LIN {X -0.070,Y -172.197,Z 547.386,A 0.000,B 0.000,C 90.000,E1 249.571} C_DIS
LIN {X -0.092,Y -171.671,Z 547.382,A 0.000,B 0.000,C 90.000,E1 248.720} C_DIS
LIN {X -0.100,Y -167.896,Z 547.358,A 0.000,B 0.000,C 90.000,E1 244.409} C_DIS
LIN {X 0.066,Y -166.635,Z 547.348,A 0.000,B 0.000,C 90.000,E1 242.615} C_DIS
LIN {X -0.026,Y -162.621,Z 547.324,A 0.000,B 0.000,C 90.000,E1 238.280} C_DIS
LIN {X 0.033,Y -161.308,Z 547.314,A 0.000,B 0.000,C 90.000,E1 236.501} C_DIS
LIN {X -0.057,Y -157.304,Z 547.289,A 0.000,B 0.000,C 90.000,E1 232.110} C_DIS
LIN {X 0.095,Y -155.281,Z 547.275,A 0.000,B 0.000,C 90.000,E1 229.380} C_DIS
LIN {X 0.023,Y -151.646,Z 547.250,A 0.000,B 0.000,C 90.000,E1 224.919} C_DIS
LIN {X -0.040,Y -150.514,Z 547.240,A 0.000,B 0.000,C 90.000,E1 223.137} C_DIS
LIN {X -0.016,Y -147.239,Z 547.214,A 0.000,B 0.000,C 90.000,E1 218.588} C_DIS
LIN {X -0.050,Y -145.263,Z 547.194,A 0.000,B 0.000,C 90.000,E1 214.945} C_DIS
LIN {X -0.016,Y -142.373,Z 547.163,A 0.000,B 0.000,C 90.000,E1 209.411} C_DIS
LIN {X -0.021,Y -141.757,Z 547.153,A 0.000,B 0.000,C 90.000,E1 207.564} C_DIS
LIN {X 0.030,Y -139.498,Z 547.117,A 0.000,B 0.000,C 90.000,E1 201.046} C_DIS
LIN {X 0.066,Y -139.004,Z 547.101,A 0.000,B 0.000,C 90.000,E1 198.236} C_DIS
LIN {X 0.023,Y -138.339,Z 547.055,A 0.000,B 0.000,C 90.000,E1 189.849} C_DIS
LIN {X 0.045,Y -139.406,Z 547.008,A 0.000,B 0.000,C 90.000,E1 181.432} C_DIS
LIN {X -0.041,Y -141.314,Z 546.972,A 0.000,B 0.000,C 90.000,E1 174.951} C_DIS
LIN {X 0.057,Y -142.673,Z 546.956,A 0.000,B 0.000,C 90.000,E1 172.129} C_DIS
LIN {X 0.038,Y -145.026,Z 546.931,A 0.000,B 0.000,C 90.000,E1 167.521} C_DIS
LIN {X -0.005,Y -147.652,Z 546.910,A 0.000,B 0.000,C 90.000,E1 163.866} C_DIS
LIN {X -0.071,Y -150.288,Z 546.890,A 0.000,B 0.000,C 90.000,E1 160.242} C_DIS
LIN {X -0.058,Y -153.695,Z 546.870,A 0.000,B 0.000,C 90.000,E1 156.613} C_DIS
LIN {X -0.003,Y -157.109,Z 546.850,A 0.000,B 0.000,C 90.000,E1 152.999} C_DIS
LIN {X 0.074,Y -161.250,Z 546.830,A 0.000,B 0.000,C 90.000,E1 149.410} C_DIS
LIN {X 0.020,Y -163.336,Z 546.820,A 0.000,B 0.000,C 90.000,E1 147.661} C_DIS
LIN {X 0.026,Y -167.791,Z 546.801,A 0.000,B 0.000,C 90.000,E1 144.149} C_DIS
LIN {X 0.041,Y -171.605,Z 546.786,A 0.000,B 0.000,C 90.000,E1 141.537} C_DIS
LIN {X 0.090,Y -176.559,Z 546.767,A 0.000,B 0.000,C 90.000,E1 138.081} C_DIS
LIN {X -0.036,Y -180.857,Z 546.753,A 0.000,B 0.000,C 90.000,E1 135.567} C_DIS
LIN {X -0.052,Y -186.270,Z 546.734,A 0.000,B 0.000,C 90.000,E1 132.204} C_DIS
LIN {X 0.015,Y -191.369,Z 546.719,A 0.000,B 0.000,C 90.000,E1 129.402} C_DIS
LIN {X -0.035,Y -191.935,Z 546.717,A 0.000,B 0.000,C 90.000,E1 129.072} C_DIS
LIN {X 0.095,Y -289.045,Z 546.717,A 0.000,B 0.000,C 90.000,E1 129.036} C_DIS
LIN {X -0.010,Y -290.435,Z 546.717,A 0.000,B 0.000,C 90.000,E1 129.036} C_DIS
LIN {X 0.173,Y -294.486,Z 546.716,A 0.000,B 0.000,C 90.000,E1 128.830} C_DIS
LIN {X 0.062,Y -297.700,Z 546.714,A 0.000,B 0.000,C 90.000,E1 128.588} C_DIS
LIN {X 0.115,Y -301.387,Z 546.712,A 0.000,B 0.000,C 90.000,E1 128.096} C_DIS
LIN {X -0.126,Y -303.164,Z 546.710,A 0.000,B 0.000,C 90.000,E1 127.810} C_DIS
LIN {X 0.057,Y -304.555,Z 546.708,A 0.000,B 0.000,C 90.000,E1 127.443} C_DIS
LIN {X 0.012,Y -308.418,Z 546.701,A 0.000,B 0.000,C 90.000,E1 126.137} C_DIS
LIN {X 0.078,Y -318.623,Z 546.683,A 0.000,B 0.000,C 90.000,E1 122.880} C_DIS
LIN {X 0.153,Y -329.135,Z 546.667,A 0.000,B 0.000,C 90.000,E1 120.001} C_DIS
LIN {X 0.045,Y -341.016,Z 546.651,A 0.000,B 0.000,C 90.000,E1 117.206} C_DIS
LIN {X -0.031,Y -354.367,Z 546.636,A 0.000,B 0.000,C 90.000,E1 114.463} C_DIS
LIN {X -0.113,Y -367.569,Z 546.623,A 0.000,B 0.000,C 90.000,E1 112.078} C_DIS
LIN {X 0.070,Y -382.126,Z 546.609,A 0.000,B 0.000,C 90.000,E1 109.704} C_DIS
LIN {X 0.149,Y -398.143,Z 546.597,A 0.000,B 0.000,C 90.000,E1 107.402} C_DIS
LIN {X -0.002,Y -415.738,Z 546.584,A 0.000,B 0.000,C 90.000,E1 105.190} C_DIS
LIN {X 0.088,Y -435.005,Z 546.572,A 0.000,B 0.000,C 90.000,E1 103.008} C_DIS
LIN {X -0.087,Y -455.210,Z 546.561,A 0.000,B 0.000,C 90.000,E1 101.007} C_DIS
LIN {X -0.092,Y -475.919,Z 546.551,A 0.000,B 0.000,C 90.000,E1 99.151} C_DIS
LIN {X 0.019,Y -477.987,Z 546.550,A 0.000,B 0.000,C 90.000,E1 98.916} C_DIS
LIN {X -0.115,Y -479.747,Z 546.548,A 0.000,B 0.000,C 90.000,E1 98.681} C_DIS
LIN {X 0.155,Y -481.069,Z 546.547,A 0.000,B 0.000,C 90.000,E1 98.398} C_DIS
LIN {X -0.161,Y -482.719,Z 546.544,A 0.000,B 0.000,C 90.000,E1 97.936} C_DIS
LIN {X 0.071,Y -483.299,Z 546.541,A 0.000,B 0.000,C 90.000,E1 97.409} C_DIS
LIN {X 0.248,Y -482.905,Z 546.538,A 0.000,B 0.000,C 90.000,E1 96.891} C_DIS
LIN {X -0.050,Y -481.476,Z 546.536,A 0.000,B 0.000,C 90.000,E1 96.429} C_DIS
LIN {X -0.225,Y -480.299,Z 546.534,A 0.000,B 0.000,C 90.000,E1 96.201} C_DIS
LIN {X 0.127,Y -478.728,Z 546.533,A 0.000,B 0.000,C 90.000,E1 95.910} C_DIS
LIN {X -0.090,Y -461.364,Z 546.520,A 0.000,B 0.000,C 90.000,E1 93.669} C_DIS
LIN {X -0.033,Y -450.979,Z 546.512,A 0.000,B 0.000,C 90.000,E1 92.121} C_DIS
LIN {X -0.051,Y -437.218,Z 546.499,A 0.000,B 0.000,C 90.000,E1 89.771} C_DIS
LIN {X -0.127,Y -429.303,Z 546.491,A 0.000,B 0.000,C 90.000,E1 88.453} C_DIS
LIN {X 0.048,Y -416.530,Z 546.479,A 0.000,B 0.000,C 90.000,E1 86.274} C_DIS
LIN {X -0.049,Y -403.962,Z 546.467,A 0.000,B 0.000,C 90.000,E1 84.090} C_DIS
LIN {X 0.042,Y -391.625,Z 546.455,A 0.000,B 0.000,C 90.000,E1 81.837} C_DIS
LIN {X -0.102,Y -382.389,Z 546.445,A 0.000,B 0.000,C 90.000,E1 80.151} C_DIS
LIN {X -0.027,Y -371.645,Z 546.434,A 0.000,B 0.000,C 90.000,E1 78.117} C_DIS
LIN {X -0.023,Y -358.447,Z 546.419,A 0.000,B 0.000,C 90.000,E1 75.463} C_DIS
LIN {X -0.192,Y -348.165,Z 546.406,A 0.000,B 0.000,C 90.000,E1 73.087} C_DIS
LIN {X 0.034,Y -340.049,Z 546.394,A 0.000,B 0.000,C 90.000,E1 70.913} C_DIS
LIN {X 0.097,Y -327.539,Z 546.373,A 0.000,B 0.000,C 90.000,E1 67.177} C_DIS
LIN {X 0.041,Y -317.890,Z 546.356,A 0.000,B 0.000,C 90.000,E1 64.024} C_DIS
LIN {X 0.004,Y -310.442,Z 546.341,A 0.000,B 0.000,C 90.000,E1 61.463} C_DIS
LIN {X -0.043,Y -302.984,Z 546.327,A 0.000,B 0.000,C 90.000,E1 58.869} C_DIS
LIN {X 0.061,Y -294.026,Z 546.309,A 0.000,B 0.000,C 90.000,E1 55.548} C_DIS
LIN {X -0.050,Y -287.193,Z 546.294,A 0.000,B 0.000,C 90.000,E1 52.889} C_DIS
LIN {X -0.004,Y -282.059,Z 546.282,A 0.000,B 0.000,C 90.000,E1 50.848} C_DIS
LIN {X 0.118,Y -276.452,Z 546.271,A 0.000,B 0.000,C 90.000,E1 48.771} C_DIS
LIN {X 0.117,Y -272.330,Z 546.263,A 0.000,B 0.000,C 90.000,E1 47.391} C_DIS
LIN {X 0.127,Y -266.837,Z 546.254,A 0.000,B 0.000,C 90.000,E1 45.648} C_DIS
LIN {X 0.083,Y -259.769,Z 546.242,A 0.000,B 0.000,C 90.000,E1 43.542} C_DIS
LIN {X 0.002,Y -248.281,Z 546.222,A 0.000,B 0.000,C 90.000,E1 39.967} C_DIS
LIN {X 0.028,Y -238.665,Z 546.204,A 0.000,B 0.000,C 90.000,E1 36.664} C_DIS
LIN {X -0.074,Y -230.808,Z 546.187,A 0.000,B 0.000,C 90.000,E1 33.706} C_DIS
LIN {X -0.045,Y -223.755,Z 546.170,A 0.000,B 0.000,C 90.000,E1 30.669} C_DIS
LIN {X -0.028,Y -217.536,Z 546.153,A 0.000,B 0.000,C 90.000,E1 27.590} C_DIS
LIN {X 0.020,Y -212.107,Z 546.136,A 0.000,B 0.000,C 90.000,E1 24.463} C_DIS
LIN {X -0.036,Y -206.520,Z 546.114,A 0.000,B 0.000,C 90.000,E1 20.536} C_DIS
LIN {X -0.048,Y -202.027,Z 546.092,A 0.000,B 0.000,C 90.000,E1 16.551} C_DIS
LIN {X -0.081,Y -198.706,Z 546.070,A 0.000,B 0.000,C 90.000,E1 12.535} C_DIS
LIN {X -0.008,Y -195.844,Z 546.038,A 0.000,B 0.000,C 90.000,E1 6.834} C_DIS
LIN {X -0.024,Y -195.870,Z 545.979,A 0.000,B 0.000,C 90.000,E1 356.274} C_DIS
LIN {X 0.050,Y -198.724,Z 545.948,A 0.000,B 0.000,C 90.000,E1 350.557} C_DIS
LIN {X 0.079,Y -202.621,Z 545.921,A 0.000,B 0.000,C 90.000,E1 345.700} C_DIS
LIN {X 0.017,Y -206.754,Z 545.898,A 0.000,B 0.000,C 90.000,E1 341.710} C_DIS
LIN {X 0.012,Y -211.728,Z 545.876,A 0.000,B 0.000,C 90.000,E1 337.741} C_DIS
LIN {X -0.006,Y -217.254,Z 545.855,A 0.000,B 0.000,C 90.000,E1 333.819} C_DIS
LIN {X 0.067,Y -223.354,Z 545.833,A 0.000,B 0.000,C 90.000,E1 329.921} C_DIS
LIN {X 0.085,Y -230.113,Z 545.812,A 0.000,B 0.000,C 90.000,E1 326.087} C_DIS
LIN {X -0.001,Y -235.917,Z 545.795,A 0.000,B 0.000,C 90.000,E1 323.084} C_DIS
LIN {X -0.111,Y -243.607,Z 545.774,A 0.000,B 0.000,C 90.000,E1 319.380} C_DIS
LIN {X 0.151,Y -252.265,Z 545.754,A 0.000,B 0.000,C 90.000,E1 315.648} C_DIS
LIN {X -0.011,Y -262.199,Z 545.734,A 0.000,B 0.000,C 90.000,E1 312.081} C_DIS
LIN {X 0.031,Y -273.518,Z 545.714,A 0.000,B 0.000,C 90.000,E1 308.543} C_DIS
LIN {X -0.026,Y -286.116,Z 545.695,A 0.000,B 0.000,C 90.000,E1 305.105} C_DIS
LIN {X 0.059,Y -300.199,Z 545.676,A 0.000,B 0.000,C 90.000,E1 301.720} C_DIS
LIN {X 0.124,Y -312.274,Z 545.662,A 0.000,B 0.000,C 90.000,E1 299.077} C_DIS
LIN {X -0.142,Y -326.845,Z 545.646,A 0.000,B 0.000,C 90.000,E1 296.232} C_DIS
LIN {X -0.113,Y -339.476,Z 545.633,A 0.000,B 0.000,C 90.000,E1 294.027} C_DIS
LIN {X 0.048,Y -351.407,Z 545.623,A 0.000,B 0.000,C 90.000,E1 292.153} C_DIS
LIN {X -0.019,Y -368.800,Z 545.610,A 0.000,B 0.000,C 90.000,E1 289.758} C_DIS
LIN {X 0.098,Y -385.146,Z 545.598,A 0.000,B 0.000,C 90.000,E1 287.692} C_DIS
LIN {X -0.046,Y -402.080,Z 545.587,A 0.000,B 0.000,C 90.000,E1 285.717} C_DIS
LIN {X -0.142,Y -416.797,Z 545.578,A 0.000,B 0.000,C 90.000,E1 284.064} C_DIS
LIN {X -0.154,Y -428.707,Z 545.570,A 0.000,B 0.000,C 90.000,E1 282.703} C_DIS
LIN {X 0.133,Y -437.908,Z 545.565,A 0.000,B 0.000,C 90.000,E1 281.591} C_DIS
LIN {X -0.204,Y -444.480,Z 545.560,A 0.000,B 0.000,C 90.000,E1 280.838} C_DIS
LIN {X -0.161,Y -452.677,Z 545.554,A 0.000,B 0.000,C 90.000,E1 279.782} C_DIS
LIN {X -0.175,Y -460.261,Z 545.548,A 0.000,B 0.000,C 90.000,E1 278.746} C_DIS
LIN {X 0.149,Y -465.527,Z 545.544,A 0.000,B 0.000,C 90.000,E1 277.936} C_DIS
LIN {X 0.053,Y -470.288,Z 545.540,A 0.000,B 0.000,C 90.000,E1 277.182} C_DIS
LIN {X -0.001,Y -474.504,Z 545.536,A 0.000,B 0.000,C 90.000,E1 276.429} C_DIS
LIN {X -0.077,Y -478.274,Z 545.531,A 0.000,B 0.000,C 90.000,E1 275.682} C_DIS
LIN {X 0.068,Y -480.405,Z 545.529,A 0.000,B 0.000,C 90.000,E1 275.163} C_DIS
LIN {X 0.225,Y -482.231,Z 545.526,A 0.000,B 0.000,C 90.000,E1 274.645} C_DIS
LIN {X -0.129,Y -483.769,Z 545.523,A 0.000,B 0.000,C 90.000,E1 274.188} C_DIS
LIN {X 0.044,Y -485.000,Z 545.520,A 0.000,B 0.000,C 90.000,E1 273.669} C_DIS
LIN {X 0.196,Y -485.831,Z 545.518,A 0.000,B 0.000,C 90.000,E1 273.154} C_DIS
LIN {X -0.104,Y -486.404,Z 545.515,A 0.000,B 0.000,C 90.000,E1 272.694} C_DIS
LIN {X 0.064,Y -486.626,Z 545.512,A 0.000,B 0.000,C 90.000,E1 272.178} C_DIS
LIN {X -0.234,Y -486.498,Z 545.509,A 0.000,B 0.000,C 90.000,E1 271.718} C_DIS
LIN {X -0.061,Y -485.933,Z 545.507,A 0.000,B 0.000,C 90.000,E1 271.203} C_DIS
LIN {X 0.112,Y -484.982,Z 545.504,A 0.000,B 0.000,C 90.000,E1 270.688} C_DIS
LIN {X -0.202,Y -483.464,Z 545.501,A 0.000,B 0.000,C 90.000,E1 270.229} C_DIS
LIN {X -0.036,Y -481.307,Z 545.498,A 0.000,B 0.000,C 90.000,E1 269.714} C_DIS
LIN {X 0.119,Y -478.472,Z 545.496,A 0.000,B 0.000,C 90.000,E1 269.198} C_DIS
LIN {X -0.053,Y -476.758,Z 545.494,A 0.000,B 0.000,C 90.000,E1 268.969} C_DIS
LIN {X -0.224,Y -474.771,Z 545.493,A 0.000,B 0.000,C 90.000,E1 268.740} C_DIS
LIN {X -0.110,Y -470.060,Z 545.490,A 0.000,B 0.000,C 90.000,E1 268.224} C_DIS
LIN {X 0.194,Y -467.224,Z 545.489,A 0.000,B 0.000,C 90.000,E1 267.936} C_DIS
LIN {X 0.015,Y -464.003,Z 545.487,A 0.000,B 0.000,C 90.000,E1 267.707} C_DIS
LIN {X 0.162,Y -460.906,Z 545.486,A 0.000,B 0.000,C 90.000,E1 267.478} C_DIS
LIN {X -0.161,Y -454.171,Z 545.484,A 0.000,B 0.000,C 90.000,E1 267.135} C_DIS
LIN {X 0.082,Y -447.074,Z 545.482,A 0.000,B 0.000,C 90.000,E1 266.788} C_DIS
LIN {X -0.182,Y -439.758,Z 545.481,A 0.000,B 0.000,C 90.000,E1 266.560} C_DIS
LIN {X -0.050,Y -431.608,Z 545.480,A 0.000,B 0.000,C 90.000,E1 266.331} C_DIS
LIN {X 0.058,Y -423.111,Z 545.479,A 0.000,B 0.000,C 90.000,E1 266.159} C_DIS
LIN {X 0.085,Y -412.497,Z 545.478,A 0.000,B 0.000,C 90.000,E1 266.045} C_DIS
LIN {X -0.072,Y -404.407,Z 545.478,A 0.000,B 0.000,C 90.000,E1 266.045} C_DIS
LIN {X -0.066,Y -180.921,Z 545.478,A 0.000,B 0.000,C 90.000,E1 266.045} C_DIS
LIN {X -0.026,Y -180.862,Z 545.472,A 0.000,B 0.000,C 90.000,E1 265.008} C_DIS
LIN {X 0.054,Y -178.917,Z 545.443,A 0.000,B 0.000,C 90.000,E1 259.746} C_DIS
LIN {X -0.037,Y -175.963,Z 545.415,A 0.000,B 0.000,C 90.000,E1 254.685} C_DIS
LIN {X 0.079,Y -175.438,Z 545.410,A 0.000,B 0.000,C 90.000,E1 253.795} C_DIS
LIN {X -0.080,Y -172.196,Z 545.386,A 0.000,B 0.000,C 90.000,E1 249.571} C_DIS
LIN {X -0.101,Y -171.669,Z 545.382,A 0.000,B 0.000,C 90.000,E1 248.720} C_DIS
LIN {X 0.042,Y -167.894,Z 545.358,A 0.000,B 0.000,C 90.000,E1 244.357} C_DIS
LIN {X 0.057,Y -166.632,Z 545.348,A 0.000,B 0.000,C 90.000,E1 242.615} C_DIS
LIN {X -0.035,Y -162.618,Z 545.324,A 0.000,B 0.000,C 90.000,E1 238.280} C_DIS
LIN {X 0.023,Y -161.304,Z 545.314,A 0.000,B 0.000,C 90.000,E1 236.501} C_DIS
LIN {X -0.067,Y -157.302,Z 545.289,A 0.000,B 0.000,C 90.000,E1 232.110} C_DIS
LIN {X 0.086,Y -155.278,Z 545.275,A 0.000,B 0.000,C 90.000,E1 229.380} C_DIS
LIN {X 0.014,Y -151.643,Z 545.250,A 0.000,B 0.000,C 90.000,E1 224.919} C_DIS
LIN {X -0.049,Y -150.512,Z 545.240,A 0.000,B 0.000,C 90.000,E1 223.137} C_DIS
LIN {X -0.025,Y -147.237,Z 545.214,A 0.000,B 0.000,C 90.000,E1 218.588} C_DIS
LIN {X 0.060,Y -145.260,Z 545.194,A 0.000,B 0.000,C 90.000,E1 214.898} C_DIS
LIN {X -0.025,Y -142.371,Z 545.163,A 0.000,B 0.000,C 90.000,E1 209.411} C_DIS
LIN {X -0.030,Y -141.756,Z 545.153,A 0.000,B 0.000,C 90.000,E1 207.564} C_DIS
LIN {X 0.021,Y -139.497,Z 545.117,A 0.000,B 0.000,C 90.000,E1 201.046} C_DIS
LIN {X 0.058,Y -139.003,Z 545.101,A 0.000,B 0.000,C 90.000,E1 198.236} C_DIS
LIN {X 0.014,Y -138.339,Z 545.055,A 0.000,B 0.000,C 90.000,E1 189.849} C_DIS
LIN {X 0.036,Y -139.406,Z 545.008,A 0.000,B 0.000,C 90.000,E1 181.432} C_DIS
LIN {X -0.050,Y -141.316,Z 544.972,A 0.000,B 0.000,C 90.000,E1 174.951} C_DIS
LIN {X 0.049,Y -142.675,Z 544.956,A 0.000,B 0.000,C 90.000,E1 172.129} C_DIS
LIN {X 0.029,Y -145.028,Z 544.931,A 0.000,B 0.000,C 90.000,E1 167.521} C_DIS
LIN {X -0.014,Y -147.655,Z 544.910,A 0.000,B 0.000,C 90.000,E1 163.866} C_DIS
LIN {X 0.062,Y -150.292,Z 544.890,A 0.000,B 0.000,C 90.000,E1 160.188} C_DIS
LIN {X -0.067,Y -153.699,Z 544.870,A 0.000,B 0.000,C 90.000,E1 156.613} C_DIS
LIN {X -0.012,Y -157.113,Z 544.850,A 0.000,B 0.000,C 90.000,E1 152.999} C_DIS
LIN {X 0.064,Y -161.255,Z 544.830,A 0.000,B 0.000,C 90.000,E1 149.410} C_DIS
LIN {X -0.008,Y -164.373,Z 544.815,A 0.000,B 0.000,C 90.000,E1 146.786} C_DIS
LIN {X -0.021,Y -169.047,Z 544.796,A 0.000,B 0.000,C 90.000,E1 143.290} C_DIS
LIN {X 0.032,Y -171.609,Z 544.786,A 0.000,B 0.000,C 90.000,E1 141.537} C_DIS
LIN {X 0.080,Y -176.565,Z 544.767,A 0.000,B 0.000,C 90.000,E1 138.081} C_DIS
LIN {X -0.046,Y -180.863,Z 544.753,A 0.000,B 0.000,C 90.000,E1 135.567} C_DIS
LIN {X -0.063,Y -186.276,Z 544.734,A 0.000,B 0.000,C 90.000,E1 132.204} C_DIS
LIN {X 0.003,Y -191.374,Z 544.719,A 0.000,B 0.000,C 90.000,E1 129.402} C_DIS
LIN {X 0.026,Y -191.964,Z 544.717,A 0.000,B 0.000,C 90.000,E1 129.036} C_DIS
LIN {X 0.006,Y -288.546,Z 544.717,A 0.000,B 0.000,C 90.000,E1 129.036} C_DIS
LIN {X -0.029,Y -289.471,Z 544.717,A 0.000,B 0.000,C 90.000,E1 129.036} C_DIS
LIN {X 0.156,Y -294.233,Z 544.716,A 0.000,B 0.000,C 90.000,E1 128.830} C_DIS
LIN {X 0.062,Y -297.157,Z 544.715,A 0.000,B 0.000,C 90.000,E1 128.624} C_DIS
LIN {X 0.018,Y -300.901,Z 544.712,A 0.000,B 0.000,C 90.000,E1 128.177} C_DIS
LIN {X -0.020,Y -302.779,Z 544.710,A 0.000,B 0.000,C 90.000,E1 127.855} C_DIS
LIN {X -0.005,Y -304.248,Z 544.708,A 0.000,B 0.000,C 90.000,E1 127.523} C_DIS
LIN {X -0.032,Y -306.343,Z 544.705,A 0.000,B 0.000,C 90.000,E1 126.870} C_DIS
LIN {X 0.149,Y -316.216,Z 544.687,A 0.000,B 0.000,C 90.000,E1 123.579} C_DIS
LIN {X 0.050,Y -326.408,Z 544.671,A 0.000,B 0.000,C 90.000,E1 120.718} C_DIS
LIN {X 0.013,Y -337.944,Z 544.655,A 0.000,B 0.000,C 90.000,E1 117.897} C_DIS
LIN {X -0.160,Y -350.921,Z 544.640,A 0.000,B 0.000,C 90.000,E1 115.155} C_DIS
LIN {X 0.006,Y -363.767,Z 544.626,A 0.000,B 0.000,C 90.000,E1 112.717} C_DIS
LIN {X 0.016,Y -377.939,Z 544.613,A 0.000,B 0.000,C 90.000,E1 110.355} C_DIS
LIN {X -0.026,Y -393.541,Z 544.600,A 0.000,B 0.000,C 90.000,E1 108.055} C_DIS
LIN {X 0.091,Y -410.687,Z 544.588,A 0.000,B 0.000,C 90.000,E1 105.788} C_DIS
LIN {X 0.135,Y -429.504,Z 544.576,A 0.000,B 0.000,C 90.000,E1 103.592} C_DIS
LIN {X 0.020,Y -449.542,Z 544.564,A 0.000,B 0.000,C 90.000,E1 101.535} C_DIS
LIN {X 0.197,Y -470.144,Z 544.554,A 0.000,B 0.000,C 90.000,E1 99.613} C_DIS
LIN {X -0.175,Y -475.373,Z 544.551,A 0.000,B 0.000,C 90.000,E1 99.208} C_DIS
LIN {X -0.069,Y -477.617,Z 544.550,A 0.000,B 0.000,C 90.000,E1 98.973} C_DIS
LIN {X -0.223,Y -479.463,Z 544.548,A 0.000,B 0.000,C 90.000,E1 98.746} C_DIS
LIN {X 0.172,Y -480.860,Z 544.547,A 0.000,B 0.000,C 90.000,E1 98.454} C_DIS
LIN {X -0.147,Y -482.685,Z 544.544,A 0.000,B 0.000,C 90.000,E1 97.992} C_DIS
LIN {X 0.022,Y -483.410,Z 544.542,A 0.000,B 0.000,C 90.000,E1 97.473} C_DIS
LIN {X 0.261,Y -483.156,Z 544.539,A 0.000,B 0.000,C 90.000,E1 96.947} C_DIS
LIN {X -0.038,Y -481.887,Z 544.536,A 0.000,B 0.000,C 90.000,E1 96.486} C_DIS
LIN {X -0.213,Y -480.809,Z 544.535,A 0.000,B 0.000,C 90.000,E1 96.258} C_DIS
LIN {X 0.141,Y -479.362,Z 544.533,A 0.000,B 0.000,C 90.000,E1 95.967} C_DIS
LIN {X 0.053,Y -467.646,Z 544.525,A 0.000,B 0.000,C 90.000,E1 94.473} C_DIS
LIN {X 0.236,Y -456.621,Z 544.516,A 0.000,B 0.000,C 90.000,E1 92.922} C_DIS
LIN {X 0.201,Y -446.737,Z 544.508,A 0.000,B 0.000,C 90.000,E1 91.375} C_DIS
LIN {X 0.165,Y -436.140,Z 544.498,A 0.000,B 0.000,C 90.000,E1 89.542} C_DIS
LIN {X -0.204,Y -426.561,Z 544.489,A 0.000,B 0.000,C 90.000,E1 87.993} C_DIS
LIN {X -0.080,Y -413.840,Z 544.477,A 0.000,B 0.000,C 90.000,E1 85.812} C_DIS
LIN {X 0.166,Y -401.295,Z 544.464,A 0.000,B 0.000,C 90.000,E1 83.571} C_DIS
LIN {X 0.191,Y -390.524,Z 544.453,A 0.000,B 0.000,C 90.000,E1 81.602} C_DIS
LIN {X -0.010,Y -379.714,Z 544.442,A 0.000,B 0.000,C 90.000,E1 79.634} C_DIS
LIN {X 0.071,Y -368.956,Z 544.431,A 0.000,B 0.000,C 90.000,E1 77.589} C_DIS
LIN {X 0.087,Y -358.797,Z 544.420,A 0.000,B 0.000,C 90.000,E1 75.519} C_DIS
LIN {X 0.000,Y -349.685,Z 544.408,A 0.000,B 0.000,C 90.000,E1 73.433} C_DIS
LIN {X 0.160,Y -340.322,Z 544.394,A 0.000,B 0.000,C 90.000,E1 70.967} C_DIS
LIN {X -0.067,Y -327.793,Z 544.374,A 0.000,B 0.000,C 90.000,E1 67.283} C_DIS
LIN {X 0.052,Y -318.151,Z 544.356,A 0.000,B 0.000,C 90.000,E1 64.101} C_DIS
LIN {X -0.111,Y -310.668,Z 544.342,A 0.000,B 0.000,C 90.000,E1 61.563} C_DIS
LIN {X -0.032,Y -303.212,Z 544.327,A 0.000,B 0.000,C 90.000,E1 58.948} C_DIS
LIN {X -0.170,Y -294.218,Z 544.309,A 0.000,B 0.000,C 90.000,E1 55.674} C_DIS
LIN {X -0.038,Y -287.364,Z 544.294,A 0.000,B 0.000,C 90.000,E1 52.970} C_DIS
LIN {X 0.011,Y -282.228,Z 544.283,A 0.000,B 0.000,C 90.000,E1 50.928} C_DIS
LIN {X 0.134,Y -276.622,Z 544.272,A 0.000,B 0.000,C 90.000,E1 48.852} C_DIS
LIN {X 0.134,Y -272.512,Z 544.264,A 0.000,B 0.000,C 90.000,E1 47.472} C_DIS
LIN {X 0.028,Y -265.856,Z 544.252,A 0.000,B 0.000,C 90.000,E1 45.405} C_DIS
LIN {X 0.005,Y -257.606,Z 544.239,A 0.000,B 0.000,C 90.000,E1 42.933} C_DIS
LIN {X -0.144,Y -247.351,Z 544.221,A 0.000,B 0.000,C 90.000,E1 39.725} C_DIS
LIN {X 0.031,Y -236.771,Z 544.200,A 0.000,B 0.000,C 90.000,E1 36.011} C_DIS
LIN {X -0.057,Y -229.088,Z 544.183,A 0.000,B 0.000,C 90.000,E1 33.038} C_DIS
LIN {X -0.069,Y -222.232,Z 544.167,A 0.000,B 0.000,C 90.000,E1 30.001} C_DIS
LIN {X 0.099,Y -216.189,Z 544.149,A 0.000,B 0.000,C 90.000,E1 26.873} C_DIS
LIN {X 0.018,Y -210.991,Z 544.132,A 0.000,B 0.000,C 90.000,E1 23.770} C_DIS
LIN {X 0.044,Y -205.581,Z 544.110,A 0.000,B 0.000,C 90.000,E1 19.812} C_DIS
LIN {X -0.054,Y -201.321,Z 544.088,A 0.000,B 0.000,C 90.000,E1 15.843} C_DIS
LIN {X -0.070,Y -197.719,Z 544.061,A 0.000,B 0.000,C 90.000,E1 11.007} C_DIS
LIN {X 0.021,Y -195.148,Z 544.025,A 0.000,B 0.000,C 90.000,E1 4.473} C_DIS
LIN {X 0.077,Y -196.798,Z 543.966,A 0.000,B 0.000,C 90.000,E1 353.799} C_DIS
LIN {X 0.081,Y -199.822,Z 543.939,A 0.000,B 0.000,C 90.000,E1 348.926} C_DIS
LIN {X 0.041,Y -204.110,Z 543.912,A 0.000,B 0.000,C 90.000,E1 344.102} C_DIS
LIN {X 0.018,Y -208.595,Z 543.890,A 0.000,B 0.000,C 90.000,E1 340.115} C_DIS
LIN {X -0.042,Y -213.789,Z 543.868,A 0.000,B 0.000,C 90.000,E1 336.177} C_DIS
LIN {X 0.100,Y -219.568,Z 543.846,A 0.000,B 0.000,C 90.000,E1 332.231} C_DIS
LIN {X -0.045,Y -225.906,Z 543.824,A 0.000,B 0.000,C 90.000,E1 328.408} C_DIS
LIN {X -0.086,Y -232.920,Z 543.803,A 0.000,B 0.000,C 90.000,E1 324.609} C_DIS
LIN {X -0.006,Y -238.807,Z 543.787,A 0.000,B 0.000,C 90.000,E1 321.582} C_DIS
LIN {X -0.017,Y -246.908,Z 543.766,A 0.000,B 0.000,C 90.000,E1 317.877} C_DIS
LIN {X 0.164,Y -256.051,Z 543.746,A 0.000,B 0.000,C 90.000,E1 314.190} C_DIS
LIN {X 0.151,Y -266.562,Z 543.726,A 0.000,B 0.000,C 90.000,E1 310.620} C_DIS
LIN {X -0.009,Y -278.418,Z 543.706,A 0.000,B 0.000,C 90.000,E1 307.156} C_DIS
LIN {X 0.016,Y -290.186,Z 543.689,A 0.000,B 0.000,C 90.000,E1 304.072} C_DIS
LIN {X 0.076,Y -304.654,Z 543.671,A 0.000,B 0.000,C 90.000,E1 300.718} C_DIS
LIN {X 0.086,Y -320.167,Z 543.653,A 0.000,B 0.000,C 90.000,E1 297.462} C_DIS
LIN {X -0.181,Y -332.056,Z 543.640,A 0.000,B 0.000,C 90.000,E1 295.283} C_DIS
LIN {X -0.028,Y -345.275,Z 543.628,A 0.000,B 0.000,C 90.000,E1 293.078} C_DIS
LIN {X -0.126,Y -362.096,Z 543.615,A 0.000,B 0.000,C 90.000,E1 290.663} C_DIS
LIN {X -0.072,Y -382.817,Z 543.600,A 0.000,B 0.000,C 90.000,E1 288.000} C_DIS
LIN {X 0.120,Y -399.679,Z 543.589,A 0.000,B 0.000,C 90.000,E1 285.969} C_DIS
LIN {X -0.141,Y -416.800,Z 543.578,A 0.000,B 0.000,C 90.000,E1 284.064} C_DIS
LIN {X -0.148,Y -428.730,Z 543.570,A 0.000,B 0.000,C 90.000,E1 282.703} C_DIS
LIN {X -0.183,Y -440.193,Z 543.563,A 0.000,B 0.000,C 90.000,E1 281.366} C_DIS
LIN {X -0.187,Y -448.719,Z 543.557,A 0.000,B 0.000,C 90.000,E1 280.310} C_DIS
LIN {X -0.174,Y -456.633,Z 543.551,A 0.000,B 0.000,C 90.000,E1 279.265} C_DIS
LIN {X -0.067,Y -463.935,Z 543.546,A 0.000,B 0.000,C 90.000,E1 278.219} C_DIS
LIN {X -0.176,Y -468.886,Z 543.541,A 0.000,B 0.000,C 90.000,E1 277.466} C_DIS
LIN {X 0.162,Y -473.264,Z 543.537,A 0.000,B 0.000,C 90.000,E1 276.663} C_DIS
LIN {X 0.132,Y -477.178,Z 543.533,A 0.000,B 0.000,C 90.000,E1 275.910} C_DIS
LIN {X 0.081,Y -480.489,Z 543.529,A 0.000,B 0.000,C 90.000,E1 275.163} C_DIS
LIN {X 0.239,Y -482.284,Z 543.526,A 0.000,B 0.000,C 90.000,E1 274.645} C_DIS
LIN {X -0.116,Y -483.804,Z 543.523,A 0.000,B 0.000,C 90.000,E1 274.188} C_DIS
LIN {X 0.058,Y -485.042,Z 543.520,A 0.000,B 0.000,C 90.000,E1 273.669} C_DIS
LIN {X 0.211,Y -485.855,Z 543.518,A 0.000,B 0.000,C 90.000,E1 273.154} C_DIS
LIN {X -0.088,Y -486.408,Z 543.515,A 0.000,B 0.000,C 90.000,E1 272.694} C_DIS
LIN {X 0.080,Y -486.616,Z 543.512,A 0.000,B 0.000,C 90.000,E1 272.178} C_DIS
LIN {X -0.219,Y -486.488,Z 543.509,A 0.000,B 0.000,C 90.000,E1 271.718} C_DIS
LIN {X -0.046,Y -485.960,Z 543.507,A 0.000,B 0.000,C 90.000,E1 271.203} C_DIS
LIN {X 0.127,Y -484.981,Z 543.504,A 0.000,B 0.000,C 90.000,E1 270.688} C_DIS
LIN {X -0.186,Y -483.475,Z 543.501,A 0.000,B 0.000,C 90.000,E1 270.229} C_DIS
LIN {X -0.021,Y -481.312,Z 543.498,A 0.000,B 0.000,C 90.000,E1 269.714} C_DIS
LIN {X -0.183,Y -480.037,Z 543.497,A 0.000,B 0.000,C 90.000,E1 269.484} C_DIS
LIN {X -0.039,Y -476.772,Z 543.494,A 0.000,B 0.000,C 90.000,E1 268.969} C_DIS
LIN {X 0.085,Y -472.582,Z 543.491,A 0.000,B 0.000,C 90.000,E1 268.453} C_DIS
LIN {X -0.095,Y -470.075,Z 543.490,A 0.000,B 0.000,C 90.000,E1 268.224} C_DIS
LIN {X 0.093,Y -464.092,Z 543.487,A 0.000,B 0.000,C 90.000,E1 267.707} C_DIS
LIN {X 0.229,Y -461.040,Z 543.486,A 0.000,B 0.000,C 90.000,E1 267.478} C_DIS
LIN {X -0.096,Y -454.328,Z 543.484,A 0.000,B 0.000,C 90.000,E1 267.135} C_DIS
LIN {X 0.146,Y -447.382,Z 543.482,A 0.000,B 0.000,C 90.000,E1 266.788} C_DIS
LIN {X -0.106,Y -440.066,Z 543.481,A 0.000,B 0.000,C 90.000,E1 266.560} C_DIS
LIN {X 0.039,Y -432.372,Z 543.480,A 0.000,B 0.000,C 90.000,E1 266.331} C_DIS
LIN {X 0.146,Y -424.084,Z 543.479,A 0.000,B 0.000,C 90.000,E1 266.159} C_DIS
LIN {X 0.162,Y -414.592,Z 543.478,A 0.000,B 0.000,C 90.000,E1 266.045} C_DIS
LIN {X -0.090,Y -406.771,Z 543.478,A 0.000,B 0.000,C 90.000,E1 266.045} C_DIS
LIN {X -0.058,Y -180.921,Z 543.478,A 0.000,B 0.000,C 90.000,E1 266.045} C_DIS
LIN {X -0.001,Y -180.863,Z 543.472,A 0.000,B 0.000,C 90.000,E1 265.008} C_DIS
LIN {X 0.079,Y -178.920,Z 543.443,A 0.000,B 0.000,C 90.000,E1 259.746} C_DIS
LIN {X -0.012,Y -175.966,Z 543.415,A 0.000,B 0.000,C 90.000,E1 254.685} C_DIS
LIN {X 0.104,Y -175.446,Z 543.410,A 0.000,B 0.000,C 90.000,E1 253.795} C_DIS
LIN {X -0.056,Y -172.200,Z 543.386,A 0.000,B 0.000,C 90.000,E1 249.571} C_DIS
LIN {X -0.078,Y -171.674,Z 543.382,A 0.000,B 0.000,C 90.000,E1 248.720} C_DIS
LIN {X -0.086,Y -167.900,Z 543.358,A 0.000,B 0.000,C 90.000,E1 244.409} C_DIS
LIN {X 0.081,Y -166.639,Z 543.348,A 0.000,B 0.000,C 90.000,E1 242.615} C_DIS
LIN {X -0.013,Y -162.624,Z 543.324,A 0.000,B 0.000,C 90.000,E1 238.280} C_DIS
LIN {X 0.047,Y -161.311,Z 543.314,A 0.000,B 0.000,C 90.000,E1 236.501} C_DIS
LIN {X -0.044,Y -157.308,Z 543.289,A 0.000,B 0.000,C 90.000,E1 232.110} C_DIS
LIN {X 0.109,Y -155.286,Z 543.275,A 0.000,B 0.000,C 90.000,E1 229.380} C_DIS
LIN {X 0.036,Y -151.649,Z 543.250,A 0.000,B 0.000,C 90.000,E1 224.919} C_DIS
LIN {X -0.027,Y -150.517,Z 543.240,A 0.000,B 0.000,C 90.000,E1 223.137} C_DIS
LIN {X -0.003,Y -147.242,Z 543.214,A 0.000,B 0.000,C 90.000,E1 218.588} C_DIS
LIN {X -0.038,Y -145.266,Z 543.194,A 0.000,B 0.000,C 90.000,E1 214.945} C_DIS
LIN {X -0.004,Y -142.375,Z 543.163,A 0.000,B 0.000,C 90.000,E1 209.411} C_DIS
LIN {X 0.046,Y -141.351,Z 543.148,A 0.000,B 0.000,C 90.000,E1 206.616} C_DIS
LIN {X 0.028,Y -139.339,Z 543.112,A 0.000,B 0.000,C 90.000,E1 200.120} C_DIS
LIN {X 0.079,Y -139.006,Z 543.102,A 0.000,B 0.000,C 90.000,E1 198.236} C_DIS
LIN {X 0.035,Y -138.340,Z 543.055,A 0.000,B 0.000,C 90.000,E1 189.849} C_DIS
LIN {X 0.058,Y -139.405,Z 543.008,A 0.000,B 0.000,C 90.000,E1 181.432} C_DIS
LIN {X -0.028,Y -141.312,Z 542.972,A 0.000,B 0.000,C 90.000,E1 174.951} C_DIS
LIN {X -0.071,Y -142.671,Z 542.956,A 0.000,B 0.000,C 90.000,E1 172.186} C_DIS
LIN {X 0.050,Y -145.023,Z 542.931,A 0.000,B 0.000,C 90.000,E1 167.521} C_DIS
LIN {X 0.007,Y -147.649,Z 542.910,A 0.000,B 0.000,C 90.000,E1 163.866} C_DIS
LIN {X -0.057,Y -150.285,Z 542.890,A 0.000,B 0.000,C 90.000,E1 160.242} C_DIS
LIN {X -0.044,Y -153.690,Z 542.870,A 0.000,B 0.000,C 90.000,E1 156.613} C_DIS
LIN {X 0.011,Y -157.104,Z 542.850,A 0.000,B 0.000,C 90.000,E1 152.999} C_DIS
LIN {X -0.051,Y -161.244,Z 542.830,A 0.000,B 0.000,C 90.000,E1 149.459} C_DIS
LIN {X 0.034,Y -163.330,Z 542.820,A 0.000,B 0.000,C 90.000,E1 147.661} C_DIS
LIN {X -0.095,Y -167.784,Z 542.801,A 0.000,B 0.000,C 90.000,E1 144.196} C_DIS
LIN {X 0.056,Y -171.598,Z 542.786,A 0.000,B 0.000,C 90.000,E1 141.537} C_DIS
LIN {X 0.104,Y -176.552,Z 542.767,A 0.000,B 0.000,C 90.000,E1 138.081} C_DIS
LIN {X -0.021,Y -180.850,Z 542.753,A 0.000,B 0.000,C 90.000,E1 135.567} C_DIS
LIN {X -0.038,Y -186.261,Z 542.734,A 0.000,B 0.000,C 90.000,E1 132.204} C_DIS
LIN {X 0.026,Y -191.364,Z 542.719,A 0.000,B 0.000,C 90.000,E1 129.402} C_DIS
LIN {X -0.069,Y -192.012,Z 542.717,A 0.000,B 0.000,C 90.000,E1 129.036} C_DIS
LIN {X 0.086,Y -289.452,Z 542.717,A 0.000,B 0.000,C 90.000,E1 128.991} C_DIS
LIN {X -0.034,Y -293.751,Z 542.716,A 0.000,B 0.000,C 90.000,E1 128.874} C_DIS
LIN {X -0.037,Y -296.674,Z 542.715,A 0.000,B 0.000,C 90.000,E1 128.669} C_DIS
LIN {X -0.104,Y -300.408,Z 542.712,A 0.000,B 0.000,C 90.000,E1 128.257} C_DIS
LIN {X -0.057,Y -302.326,Z 542.711,A 0.000,B 0.000,C 90.000,E1 127.935} C_DIS
LIN {X 0.043,Y -303.831,Z 542.709,A 0.000,B 0.000,C 90.000,E1 127.604} C_DIS
LIN {X 0.000,Y -305.087,Z 542.707,A 0.000,B 0.000,C 90.000,E1 127.282} C_DIS
LIN {X -0.007,Y -316.973,Z 542.685,A 0.000,B 0.000,C 90.000,E1 123.372} C_DIS
LIN {X 0.186,Y -327.272,Z 542.669,A 0.000,B 0.000,C 90.000,E1 120.463} C_DIS
LIN {X 0.187,Y -338.918,Z 542.654,A 0.000,B 0.000,C 90.000,E1 117.641} C_DIS
LIN {X 0.045,Y -352.021,Z 542.638,A 0.000,B 0.000,C 90.000,E1 114.899} C_DIS
LIN {X -0.093,Y -364.983,Z 542.625,A 0.000,B 0.000,C 90.000,E1 112.514} C_DIS
LIN {X 0.155,Y -379.282,Z 542.612,A 0.000,B 0.000,C 90.000,E1 110.120} C_DIS
LIN {X 0.160,Y -395.021,Z 542.599,A 0.000,B 0.000,C 90.000,E1 107.819} C_DIS
LIN {X -0.070,Y -412.315,Z 542.587,A 0.000,B 0.000,C 90.000,E1 105.607} C_DIS
LIN {X 0.003,Y -431.292,Z 542.575,A 0.000,B 0.000,C 90.000,E1 103.411} C_DIS
LIN {X -0.087,Y -451.390,Z 542.563,A 0.000,B 0.000,C 90.000,E1 101.366} C_DIS
LIN {X -0.248,Y -472.038,Z 542.553,A 0.000,B 0.000,C 90.000,E1 99.500} C_DIS
LIN {X -0.049,Y -477.087,Z 542.550,A 0.000,B 0.000,C 90.000,E1 99.029} C_DIS
LIN {X -0.102,Y -479.015,Z 542.549,A 0.000,B 0.000,C 90.000,E1 98.803} C_DIS
LIN {X -0.080,Y -480.487,Z 542.548,A 0.000,B 0.000,C 90.000,E1 98.568} C_DIS
LIN {X 0.270,Y -481.687,Z 542.546,A 0.000,B 0.000,C 90.000,E1 98.276} C_DIS
LIN {X 0.075,Y -482.562,Z 542.545,A 0.000,B 0.000,C 90.000,E1 98.049} C_DIS
LIN {X -0.231,Y -483.489,Z 542.542,A 0.000,B 0.000,C 90.000,E1 97.587} C_DIS
LIN {X -0.053,Y -483.428,Z 542.539,A 0.000,B 0.000,C 90.000,E1 97.068} C_DIS
LIN {X 0.132,Y -482.372,Z 542.536,A 0.000,B 0.000,C 90.000,E1 96.549} C_DIS
LIN {X 0.011,Y -481.421,Z 542.535,A 0.000,B 0.000,C 90.000,E1 96.315} C_DIS
LIN {X -0.162,Y -480.130,Z 542.534,A 0.000,B 0.000,C 90.000,E1 96.087} C_DIS
LIN {X 0.010,Y -476.432,Z 542.531,A 0.000,B 0.000,C 90.000,E1 95.568} C_DIS
LIN {X -0.034,Y -460.979,Z 542.520,A 0.000,B 0.000,C 90.000,E1 93.555} C_DIS
LIN {X 0.016,Y -450.574,Z 542.511,A 0.000,B 0.000,C 90.000,E1 92.007} C_DIS
LIN {X -0.017,Y -436.781,Z 542.498,A 0.000,B 0.000,C 90.000,E1 89.656} C_DIS
LIN {X 0.055,Y -427.197,Z 542.489,A 0.000,B 0.000,C 90.000,E1 88.051} C_DIS
LIN {X 0.186,Y -414.468,Z 542.477,A 0.000,B 0.000,C 90.000,E1 85.869} C_DIS
LIN {X 0.042,Y -401.896,Z 542.465,A 0.000,B 0.000,C 90.000,E1 83.685} C_DIS
LIN {X 0.028,Y -391.108,Z 542.454,A 0.000,B 0.000,C 90.000,E1 81.724} C_DIS
LIN {X -0.097,Y -380.280,Z 542.443,A 0.000,B 0.000,C 90.000,E1 79.746} C_DIS
LIN {X 0.004,Y -369.490,Z 542.432,A 0.000,B 0.000,C 90.000,E1 77.701} C_DIS
LIN {X 0.004,Y -357.915,Z 542.419,A 0.000,B 0.000,C 90.000,E1 75.338} C_DIS
LIN {X -0.102,Y -348.878,Z 542.407,A 0.000,B 0.000,C 90.000,E1 73.251} C_DIS
LIN {X -0.067,Y -338.529,Z 542.392,A 0.000,B 0.000,C 90.000,E1 70.496} C_DIS
LIN {X 0.060,Y -326.170,Z 542.371,A 0.000,B 0.000,C 90.000,E1 66.741} C_DIS
LIN {X 0.090,Y -318.503,Z 542.357,A 0.000,B 0.000,C 90.000,E1 64.204} C_DIS
LIN {X 0.073,Y -310.978,Z 542.343,A 0.000,B 0.000,C 90.000,E1 61.641} C_DIS
LIN {X -0.111,Y -303.537,Z 542.328,A 0.000,B 0.000,C 90.000,E1 59.076} C_DIS
LIN {X 0.011,Y -294.496,Z 542.310,A 0.000,B 0.000,C 90.000,E1 55.754} C_DIS
LIN {X 0.142,Y -287.613,Z 542.295,A 0.000,B 0.000,C 90.000,E1 53.050} C_DIS
LIN {X 0.012,Y -282.464,Z 542.284,A 0.000,B 0.000,C 90.000,E1 51.045} C_DIS
LIN {X -0.078,Y -276.896,Z 542.272,A 0.000,B 0.000,C 90.000,E1 49.013} C_DIS
LIN {X -0.071,Y -272.801,Z 542.265,A 0.000,B 0.000,C 90.000,E1 47.634} C_DIS
LIN {X 0.020,Y -266.160,Z 542.253,A 0.000,B 0.000,C 90.000,E1 45.526} C_DIS
LIN {X -0.002,Y -257.917,Z 542.239,A 0.000,B 0.000,C 90.000,E1 43.056} C_DIS
LIN {X 0.049,Y -246.532,Z 542.219,A 0.000,B 0.000,C 90.000,E1 39.439} C_DIS
LIN {X 0.020,Y -237.025,Z 542.201,A 0.000,B 0.000,C 90.000,E1 36.137} C_DIS
LIN {X -0.066,Y -229.288,Z 542.184,A 0.000,B 0.000,C 90.000,E1 33.166} C_DIS
LIN {X -0.075,Y -222.422,Z 542.167,A 0.000,B 0.000,C 90.000,E1 30.129} C_DIS
LIN {X 0.097,Y -216.350,Z 542.150,A 0.000,B 0.000,C 90.000,E1 27.001} C_DIS
LIN {X 0.020,Y -211.133,Z 542.133,A 0.000,B 0.000,C 90.000,E1 23.898} C_DIS
LIN {X 0.052,Y -205.695,Z 542.111,A 0.000,B 0.000,C 90.000,E1 19.939} C_DIS
LIN {X -0.037,Y -201.405,Z 542.089,A 0.000,B 0.000,C 90.000,E1 15.969} C_DIS
LIN {X -0.043,Y -197.751,Z 542.062,A 0.000,B 0.000,C 90.000,E1 11.130} C_DIS
LIN {X 0.080,Y -195.132,Z 542.026,A 0.000,B 0.000,C 90.000,E1 4.588} C_DIS
LIN {X 0.075,Y -196.752,Z 541.966,A 0.000,B 0.000,C 90.000,E1 353.799} C_DIS
LIN {X 0.077,Y -199.765,Z 541.939,A 0.000,B 0.000,C 90.000,E1 348.926} C_DIS
LIN {X 0.034,Y -204.044,Z 541.912,A 0.000,B 0.000,C 90.000,E1 344.102} C_DIS
LIN {X 0.009,Y -208.532,Z 541.890,A 0.000,B 0.000,C 90.000,E1 340.115} C_DIS
LIN {X -0.053,Y -213.722,Z 541.868,A 0.000,B 0.000,C 90.000,E1 336.177} C_DIS
LIN {X 0.086,Y -219.510,Z 541.846,A 0.000,B 0.000,C 90.000,E1 332.231} C_DIS
LIN {X -0.060,Y -225.838,Z 541.824,A 0.000,B 0.000,C 90.000,E1 328.408} C_DIS
LIN {X 0.084,Y -232.866,Z 541.803,A 0.000,B 0.000,C 90.000,E1 324.562} C_DIS
LIN {X 0.108,Y -240.271,Z 541.782,A 0.000,B 0.000,C 90.000,E1 320.803} C_DIS
LIN {X -0.067,Y -248.592,Z 541.762,A 0.000,B 0.000,C 90.000,E1 317.148} C_DIS
LIN {X -0.006,Y -258.013,Z 541.742,A 0.000,B 0.000,C 90.000,E1 313.500} C_DIS
LIN {X -0.016,Y -267.681,Z 541.724,A 0.000,B 0.000,C 90.000,E1 310.297} C_DIS
LIN {X 0.067,Y -279.662,Z 541.704,A 0.000,B 0.000,C 90.000,E1 306.790} C_DIS
LIN {X -0.015,Y -290.176,Z 541.689,A 0.000,B 0.000,C 90.000,E1 304.072} C_DIS
LIN {X 0.042,Y -304.614,Z 541.671,A 0.000,B 0.000,C 90.000,E1 300.718} C_DIS
LIN {X 0.050,Y -320.130,Z 541.653,A 0.000,B 0.000,C 90.000,E1 297.462} C_DIS
LIN {X 0.081,Y -332.014,Z 541.640,A 0.000,B 0.000,C 90.000,E1 295.232} C_DIS
LIN {X -0.068,Y -345.273,Z 541.628,A 0.000,B 0.000,C 90.000,E1 293.078} C_DIS
LIN {X 0.170,Y -362.095,Z 541.615,A 0.000,B 0.000,C 90.000,E1 290.610} C_DIS
LIN {X -0.116,Y -382.844,Z 541.600,A 0.000,B 0.000,C 90.000,E1 288.000} C_DIS
LIN {X 0.073,Y -399.716,Z 541.589,A 0.000,B 0.000,C 90.000,E1 285.969} C_DIS
LIN {X 0.136,Y -416.967,Z 541.578,A 0.000,B 0.000,C 90.000,E1 284.008} C_DIS
LIN {X 0.194,Y -428.863,Z 541.570,A 0.000,B 0.000,C 90.000,E1 282.647} C_DIS
LIN {X -0.172,Y -440.322,Z 541.563,A 0.000,B 0.000,C 90.000,E1 281.355} C_DIS
LIN {X 0.179,Y -448.883,Z 541.557,A 0.000,B 0.000,C 90.000,E1 280.254} C_DIS
LIN {X 0.201,Y -456.811,Z 541.551,A 0.000,B 0.000,C 90.000,E1 279.208} C_DIS
LIN {X -0.142,Y -464.121,Z 541.546,A 0.000,B 0.000,C 90.000,E1 278.219} C_DIS
LIN {X 0.215,Y -469.050,Z 541.541,A 0.000,B 0.000,C 90.000,E1 277.409} C_DIS
LIN {X -0.062,Y -474.777,Z 541.536,A 0.000,B 0.000,C 90.000,E1 276.429} C_DIS
LIN {X -0.136,Y -478.501,Z 541.531,A 0.000,B 0.000,C 90.000,E1 275.682} C_DIS
LIN {X 0.010,Y -480.619,Z 541.529,A 0.000,B 0.000,C 90.000,E1 275.163} C_DIS
LIN {X 0.169,Y -482.405,Z 541.526,A 0.000,B 0.000,C 90.000,E1 274.645} C_DIS
LIN {X -0.185,Y -483.892,Z 541.523,A 0.000,B 0.000,C 90.000,E1 274.188} C_DIS
LIN {X -0.011,Y -485.110,Z 541.520,A 0.000,B 0.000,C 90.000,E1 273.669} C_DIS
LIN {X 0.141,Y -485.943,Z 541.518,A 0.000,B 0.000,C 90.000,E1 273.154} C_DIS
LIN {X -0.157,Y -486.433,Z 541.515,A 0.000,B 0.000,C 90.000,E1 272.694} C_DIS
LIN {X 0.011,Y -486.620,Z 541.512,A 0.000,B 0.000,C 90.000,E1 272.178} C_DIS
LIN {X 0.199,Y -486.493,Z 541.509,A 0.000,B 0.000,C 90.000,E1 271.661} C_DIS
LIN {X -0.114,Y -485.966,Z 541.507,A 0.000,B 0.000,C 90.000,E1 271.203} C_DIS
LIN {X 0.059,Y -484.966,Z 541.504,A 0.000,B 0.000,C 90.000,E1 270.688} C_DIS
LIN {X 0.230,Y -483.464,Z 541.501,A 0.000,B 0.000,C 90.000,E1 270.172} C_DIS
LIN {X -0.088,Y -481.314,Z 541.498,A 0.000,B 0.000,C 90.000,E1 269.714} C_DIS
LIN {X 0.067,Y -478.446,Z 541.496,A 0.000,B 0.000,C 90.000,E1 269.198} C_DIS
LIN {X -0.105,Y -476.745,Z 541.494,A 0.000,B 0.000,C 90.000,E1 268.969} C_DIS
LIN {X 0.018,Y -472.485,Z 541.491,A 0.000,B 0.000,C 90.000,E1 268.453} C_DIS
LIN {X -0.161,Y -469.962,Z 541.490,A 0.000,B 0.000,C 90.000,E1 268.224} C_DIS
LIN {X 0.042,Y -464.014,Z 541.487,A 0.000,B 0.000,C 90.000,E1 267.707} C_DIS
LIN {X 0.162,Y -460.923,Z 541.486,A 0.000,B 0.000,C 90.000,E1 267.478} C_DIS
LIN {X -0.160,Y -454.180,Z 541.484,A 0.000,B 0.000,C 90.000,E1 267.135} C_DIS
LIN {X 0.106,Y -447.295,Z 541.482,A 0.000,B 0.000,C 90.000,E1 266.788} C_DIS
LIN {X -0.122,Y -440.008,Z 541.481,A 0.000,B 0.000,C 90.000,E1 266.560} C_DIS
LIN {X 0.046,Y -432.411,Z 541.480,A 0.000,B 0.000,C 90.000,E1 266.331} C_DIS
LIN {X 0.152,Y -424.254,Z 541.479,A 0.000,B 0.000,C 90.000,E1 266.159} C_DIS
LIN {X 0.171,Y -414.950,Z 541.478,A 0.000,B 0.000,C 90.000,E1 266.045} C_DIS
LIN {X -0.100,Y -408.002,Z 541.478,A 0.000,B 0.000,C 90.000,E1 266.045} C_DIS
LIN {X -0.064,Y -180.921,Z 541.478,A 0.000,B 0.000,C 90.000,E1 266.045} C_DIS
LIN {X -0.008,Y -180.863,Z 541.472,A 0.000,B 0.000,C 90.000,E1 265.008} C_DIS
LIN {X 0.072,Y -178.920,Z 541.443,A 0.000,B 0.000,C 90.000,E1 259.746} C_DIS
LIN {X -0.019,Y -175.965,Z 541.415,A 0.000,B 0.000,C 90.000,E1 254.685} C_DIS
LIN {X 0.097,Y -175.443,Z 541.410,A 0.000,B 0.000,C 90.000,E1 253.795} C_DIS
LIN {X -0.063,Y -172.199,Z 541.386,A 0.000,B 0.000,C 90.000,E1 249.571} C_DIS
LIN {X -0.085,Y -171.673,Z 541.382,A 0.000,B 0.000,C 90.000,E1 248.720} C_DIS
LIN {X -0.093,Y -167.899,Z 541.358,A 0.000,B 0.000,C 90.000,E1 244.409} C_DIS
LIN {X 0.074,Y -166.637,Z 541.348,A 0.000,B 0.000,C 90.000,E1 242.615} C_DIS
LIN {X -0.019,Y -162.622,Z 541.324,A 0.000,B 0.000,C 90.000,E1 238.280} C_DIS
LIN {X 0.040,Y -161.310,Z 541.314,A 0.000,B 0.000,C 90.000,E1 236.501} C_DIS
LIN {X -0.050,Y -157.306,Z 541.289,A 0.000,B 0.000,C 90.000,E1 232.110} C_DIS
LIN {X 0.102,Y -155.284,Z 541.275,A 0.000,B 0.000,C 90.000,E1 229.380} C_DIS
LIN {X 0.030,Y -151.647,Z 541.250,A 0.000,B 0.000,C 90.000,E1 224.919} C_DIS
LIN {X -0.033,Y -150.516,Z 541.240,A 0.000,B 0.000,C 90.000,E1 223.137} C_DIS
LIN {X -0.010,Y -147.240,Z 541.214,A 0.000,B 0.000,C 90.000,E1 218.588} C_DIS
LIN {X -0.044,Y -145.265,Z 541.194,A 0.000,B 0.000,C 90.000,E1 214.945} C_DIS
LIN {X -0.010,Y -142.374,Z 541.163,A 0.000,B 0.000,C 90.000,E1 209.411} C_DIS
LIN {X 0.040,Y -141.349,Z 541.148,A 0.000,B 0.000,C 90.000,E1 206.616} C_DIS
LIN {X 0.022,Y -139.339,Z 541.112,A 0.000,B 0.000,C 90.000,E1 200.120} C_DIS
LIN {X 0.073,Y -139.005,Z 541.102,A 0.000,B 0.000,C 90.000,E1 198.236} C_DIS
LIN {X 0.029,Y -138.339,Z 541.055,A 0.000,B 0.000,C 90.000,E1 189.849} C_DIS
LIN {X 0.052,Y -139.405,Z 541.008,A 0.000,B 0.000,C 90.000,E1 181.432} C_DIS
LIN {X -0.035,Y -141.313,Z 540.972,A 0.000,B 0.000,C 90.000,E1 174.951} C_DIS
LIN {X -0.078,Y -142.672,Z 540.956,A 0.000,B 0.000,C 90.000,E1 172.186} C_DIS
LIN {X 0.044,Y -145.025,Z 540.931,A 0.000,B 0.000,C 90.000,E1 167.521} C_DIS
LIN {X 0.002,Y -147.651,Z 540.910,A 0.000,B 0.000,C 90.000,E1 163.866} C_DIS
LIN {X -0.064,Y -150.287,Z 540.890,A 0.000,B 0.000,C 90.000,E1 160.242} C_DIS
LIN {X -0.051,Y -153.693,Z 540.870,A 0.000,B 0.000,C 90.000,E1 156.613} C_DIS
LIN {X 0.004,Y -157.107,Z 540.850,A 0.000,B 0.000,C 90.000,E1 152.999} C_DIS
LIN {X -0.058,Y -161.247,Z 540.830,A 0.000,B 0.000,C 90.000,E1 149.459} C_DIS
LIN {X 0.027,Y -163.334,Z 540.820,A 0.000,B 0.000,C 90.000,E1 147.661} C_DIS
LIN {X 0.033,Y -167.788,Z 540.801,A 0.000,B 0.000,C 90.000,E1 144.149} C_DIS
LIN {X 0.049,Y -171.601,Z 540.786,A 0.000,B 0.000,C 90.000,E1 141.537} C_DIS
LIN {X 0.097,Y -176.556,Z 540.767,A 0.000,B 0.000,C 90.000,E1 138.081} C_DIS
LIN {X -0.028,Y -180.854,Z 540.753,A 0.000,B 0.000,C 90.000,E1 135.567} C_DIS
LIN {X -0.045,Y -186.266,Z 540.734,A 0.000,B 0.000,C 90.000,E1 132.204} C_DIS
LIN {X 0.017,Y -191.368,Z 540.719,A 0.000,B 0.000,C 90.000,E1 129.402} C_DIS
LIN {X 0.023,Y -192.040,Z 540.717,A 0.000,B 0.000,C 90.000,E1 128.991} C_DIS
LIN {X -0.001,Y -289.073,Z 540.717,A 0.000,B 0.000,C 90.000,E1 128.991} C_DIS
LIN {X 0.183,Y -293.427,Z 540.716,A 0.000,B 0.000,C 90.000,E1 128.830} C_DIS
LIN {X -0.096,Y -296.597,Z 540.715,A 0.000,B 0.000,C 90.000,E1 128.669} C_DIS
LIN {X -0.089,Y -300.276,Z 540.712,A 0.000,B 0.000,C 90.000,E1 128.257} C_DIS
LIN {X -0.019,Y -302.208,Z 540.711,A 0.000,B 0.000,C 90.000,E1 127.935} C_DIS
LIN {X 0.105,Y -303.726,Z 540.709,A 0.000,B 0.000,C 90.000,E1 127.604} C_DIS
LIN {X 0.061,Y -305.013,Z 540.707,A 0.000,B 0.000,C 90.000,E1 127.282} C_DIS
LIN {X 0.054,Y -316.915,Z 540.685,A 0.000,B 0.000,C 90.000,E1 123.372} C_DIS
LIN {X -0.034,Y -327.209,Z 540.669,A 0.000,B 0.000,C 90.000,E1 120.512} C_DIS
LIN {X -0.051,Y -338.849,Z 540.654,A 0.000,B 0.000,C 90.000,E1 117.692} C_DIS
LIN {X 0.108,Y -351.947,Z 540.638,A 0.000,B 0.000,C 90.000,E1 114.899} C_DIS
LIN {X -0.031,Y -364.904,Z 540.625,A 0.000,B 0.000,C 90.000,E1 112.514} C_DIS
LIN {X -0.137,Y -379.196,Z 540.612,A 0.000,B 0.000,C 90.000,E1 110.174} C_DIS
LIN {X -0.153,Y -394.929,Z 540.599,A 0.000,B 0.000,C 90.000,E1 107.873} C_DIS
LIN {X -0.006,Y -412.216,Z 540.587,A 0.000,B 0.000,C 90.000,E1 105.607} C_DIS
LIN {X 0.068,Y -431.185,Z 540.575,A 0.000,B 0.000,C 90.000,E1 103.411} C_DIS
LIN {X -0.026,Y -451.280,Z 540.563,A 0.000,B 0.000,C 90.000,E1 101.366} C_DIS
LIN {X -0.191,Y -471.927,Z 540.553,A 0.000,B 0.000,C 90.000,E1 99.500} C_DIS
LIN {X 0.008,Y -477.023,Z 540.550,A 0.000,B 0.000,C 90.000,E1 99.029} C_DIS
LIN {X -0.021,Y -478.985,Z 540.549,A 0.000,B 0.000,C 90.000,E1 98.803} C_DIS
LIN {X 0.024,Y -480.484,Z 540.548,A 0.000,B 0.000,C 90.000,E1 98.568} C_DIS
LIN {X -0.173,Y -481.724,Z 540.546,A 0.000,B 0.000,C 90.000,E1 98.341} C_DIS
LIN {X 0.179,Y -482.634,Z 540.545,A 0.000,B 0.000,C 90.000,E1 98.049} C_DIS
LIN {X -0.127,Y -483.616,Z 540.542,A 0.000,B 0.000,C 90.000,E1 97.587} C_DIS
LIN {X 0.052,Y -483.607,Z 540.539,A 0.000,B 0.000,C 90.000,E1 97.068} C_DIS
LIN {X -0.241,Y -482.605,Z 540.537,A 0.000,B 0.000,C 90.000,E1 96.606} C_DIS
LIN {X 0.118,Y -481.688,Z 540.535,A 0.000,B 0.000,C 90.000,E1 96.315} C_DIS
LIN {X -0.056,Y -480.437,Z 540.534,A 0.000,B 0.000,C 90.000,E1 96.087} C_DIS
LIN {X -0.183,Y -478.763,Z 540.532,A 0.000,B 0.000,C 90.000,E1 95.853} C_DIS
LIN {X 0.077,Y -461.260,Z 540.520,A 0.000,B 0.000,C 90.000,E1 93.555} C_DIS
LIN {X 0.129,Y -450.815,Z 540.511,A 0.000,B 0.000,C 90.000,E1 92.007} C_DIS
LIN {X 0.099,Y -436.961,Z 540.498,A 0.000,B 0.000,C 90.000,E1 89.656} C_DIS
LIN {X 0.171,Y -427.386,Z 540.489,A 0.000,B 0.000,C 90.000,E1 88.051} C_DIS
LIN {X -0.016,Y -413.083,Z 540.476,A 0.000,B 0.000,C 90.000,E1 85.641} C_DIS
LIN {X -0.027,Y -397.456,Z 540.460,A 0.000,B 0.000,C 90.000,E1 82.875} C_DIS
LIN {X -0.075,Y -386.630,Z 540.449,A 0.000,B 0.000,C 90.000,E1 80.905} C_DIS
LIN {X 0.106,Y -374.242,Z 540.437,A 0.000,B 0.000,C 90.000,E1 78.578} C_DIS
LIN {X 0.128,Y -362.216,Z 540.424,A 0.000,B 0.000,C 90.000,E1 76.228} C_DIS
LIN {X 0.014,Y -352.708,Z 540.412,A 0.000,B 0.000,C 90.000,E1 74.157} C_DIS
LIN {X 0.143,Y -341.905,Z 540.397,A 0.000,B 0.000,C 90.000,E1 71.402} C_DIS
LIN {X -0.023,Y -330.234,Z 540.378,A 0.000,B 0.000,C 90.000,E1 68.028} C_DIS
LIN {X 0.177,Y -320.487,Z 540.360,A 0.000,B 0.000,C 90.000,E1 64.845} C_DIS
LIN {X 0.062,Y -312.933,Z 540.346,A 0.000,B 0.000,C 90.000,E1 62.308} C_DIS
LIN {X -0.080,Y -305.442,Z 540.332,A 0.000,B 0.000,C 90.000,E1 59.744} C_DIS
LIN {X -0.089,Y -298.058,Z 540.317,A 0.000,B 0.000,C 90.000,E1 57.120} C_DIS
LIN {X -0.056,Y -289.326,Z 540.299,A 0.000,B 0.000,C 90.000,E1 53.783} C_DIS
LIN {X 0.023,Y -284.191,Z 540.287,A 0.000,B 0.000,C 90.000,E1 51.743} C_DIS
LIN {X 0.156,Y -280.664,Z 540.280,A 0.000,B 0.000,C 90.000,E1 50.356} C_DIS
LIN {X 0.024,Y -276.857,Z 540.272,A 0.000,B 0.000,C 90.000,E1 49.013} C_DIS
LIN {X 0.029,Y -272.755,Z 540.265,A 0.000,B 0.000,C 90.000,E1 47.634} C_DIS
LIN {X -0.072,Y -266.124,Z 540.253,A 0.000,B 0.000,C 90.000,E1 45.567} C_DIS
LIN {X 0.061,Y -259.072,Z 540.241,A 0.000,B 0.000,C 90.000,E1 43.419} C_DIS
LIN {X -0.061,Y -247.604,Z 540.221,A 0.000,B 0.000,C 90.000,E1 39.850} C_DIS
LIN {X -0.035,Y -236.985,Z 540.201,A 0.000,B 0.000,C 90.000,E1 36.171} C_DIS
LIN {X 0.015,Y -229.237,Z 540.184,A 0.000,B 0.000,C 90.000,E1 33.166} C_DIS
LIN {X 0.002,Y -222.386,Z 540.167,A 0.000,B 0.000,C 90.000,E1 30.129} C_DIS
LIN {X -0.022,Y -216.317,Z 540.150,A 0.000,B 0.000,C 90.000,E1 27.052} C_DIS
LIN {X -0.101,Y -211.109,Z 540.133,A 0.000,B 0.000,C 90.000,E1 23.951} C_DIS
LIN {X -0.072,Y -205.677,Z 540.111,A 0.000,B 0.000,C 90.000,E1 19.993} C_DIS
LIN {X 0.029,Y -201.405,Z 540.089,A 0.000,B 0.000,C 90.000,E1 15.969} C_DIS
LIN {X 0.023,Y -197.724,Z 540.062,A 0.000,B 0.000,C 90.000,E1 11.130} C_DIS
LIN {X -0.051,Y -195.103,Z 540.026,A 0.000,B 0.000,C 90.000,E1 4.645} C_DIS
LIN {X 0.073,Y -196.703,Z 539.966,A 0.000,B 0.000,C 90.000,E1 353.799} C_DIS
LIN {X 0.073,Y -199.689,Z 539.939,A 0.000,B 0.000,C 90.000,E1 348.926} C_DIS
LIN {X 0.027,Y -203.963,Z 539.912,A 0.000,B 0.000,C 90.000,E1 344.102} C_DIS
LIN {X -0.001,Y -208.449,Z 539.890,A 0.000,B 0.000,C 90.000,E1 340.115} C_DIS
LIN {X -0.066,Y -213.648,Z 539.868,A 0.000,B 0.000,C 90.000,E1 336.177} C_DIS
LIN {X 0.071,Y -219.440,Z 539.846,A 0.000,B 0.000,C 90.000,E1 332.231} C_DIS
LIN {X -0.079,Y -225.781,Z 539.824,A 0.000,B 0.000,C 90.000,E1 328.408} C_DIS
LIN {X 0.063,Y -232.799,Z 539.803,A 0.000,B 0.000,C 90.000,E1 324.562} C_DIS
LIN {X 0.085,Y -240.211,Z 539.782,A 0.000,B 0.000,C 90.000,E1 320.803} C_DIS
LIN {X -0.093,Y -248.547,Z 539.762,A 0.000,B 0.000,C 90.000,E1 317.148} C_DIS
LIN {X -0.034,Y -257.982,Z 539.742,A 0.000,B 0.000,C 90.000,E1 313.500} C_DIS
LIN {X -0.046,Y -267.676,Z 539.724,A 0.000,B 0.000,C 90.000,E1 310.297} C_DIS
LIN {X 0.035,Y -279.660,Z 539.704,A 0.000,B 0.000,C 90.000,E1 306.790} C_DIS
LIN {X -0.049,Y -290.166,Z 539.689,A 0.000,B 0.000,C 90.000,E1 304.072} C_DIS
LIN {X 0.008,Y -304.570,Z 539.671,A 0.000,B 0.000,C 90.000,E1 300.718} C_DIS
LIN {X 0.013,Y -320.094,Z 539.653,A 0.000,B 0.000,C 90.000,E1 297.462} C_DIS
LIN {X 0.182,Y -331.987,Z 539.640,A 0.000,B 0.000,C 90.000,E1 295.207} C_DIS
LIN {X -0.113,Y -343.295,Z 539.630,A 0.000,B 0.000,C 90.000,E1 293.387} C_DIS
LIN {X 0.025,Y -357.723,Z 539.618,A 0.000,B 0.000,C 90.000,E1 291.227} C_DIS
LIN {X 0.206,Y -380.484,Z 539.602,A 0.000,B 0.000,C 90.000,E1 288.236} C_DIS
LIN {X 0.025,Y -399.748,Z 539.589,A 0.000,B 0.000,C 90.000,E1 285.969} C_DIS
LIN {X 0.086,Y -417.023,Z 539.578,A 0.000,B 0.000,C 90.000,E1 284.008} C_DIS
LIN {X 0.079,Y -429.031,Z 539.570,A 0.000,B 0.000,C 90.000,E1 282.647} C_DIS
LIN {X 0.143,Y -440.482,Z 539.563,A 0.000,B 0.000,C 90.000,E1 281.299} C_DIS
LIN {X 0.063,Y -449.095,Z 539.557,A 0.000,B 0.000,C 90.000,E1 280.254} C_DIS
LIN {X 0.086,Y -457.036,Z 539.551,A 0.000,B 0.000,C 90.000,E1 279.208} C_DIS
LIN {X 0.203,Y -464.333,Z 539.545,A 0.000,B 0.000,C 90.000,E1 278.163} C_DIS
LIN {X 0.100,Y -469.237,Z 539.541,A 0.000,B 0.000,C 90.000,E1 277.409} C_DIS
LIN {X -0.026,Y -473.611,Z 539.537,A 0.000,B 0.000,C 90.000,E1 276.663} C_DIS
LIN {X -0.053,Y -477.502,Z 539.533,A 0.000,B 0.000,C 90.000,E1 275.910} C_DIS
LIN {X -0.103,Y -480.803,Z 539.529,A 0.000,B 0.000,C 90.000,E1 275.163} C_DIS
LIN {X 0.057,Y -482.537,Z 539.526,A 0.000,B 0.000,C 90.000,E1 274.645} C_DIS
LIN {X 0.186,Y -483.992,Z 539.523,A 0.000,B 0.000,C 90.000,E1 274.131} C_DIS
LIN {X -0.123,Y -485.188,Z 539.520,A 0.000,B 0.000,C 90.000,E1 273.669} C_DIS
LIN {X 0.031,Y -485.986,Z 539.518,A 0.000,B 0.000,C 90.000,E1 273.154} C_DIS
LIN {X 0.218,Y -486.473,Z 539.515,A 0.000,B 0.000,C 90.000,E1 272.636} C_DIS
LIN {X -0.100,Y -486.672,Z 539.512,A 0.000,B 0.000,C 90.000,E1 272.178} C_DIS
LIN {X 0.089,Y -486.502,Z 539.509,A 0.000,B 0.000,C 90.000,E1 271.661} C_DIS
LIN {X -0.224,Y -485.953,Z 539.507,A 0.000,B 0.000,C 90.000,E1 271.203} C_DIS
LIN {X -0.050,Y -484.950,Z 539.504,A 0.000,B 0.000,C 90.000,E1 270.688} C_DIS
LIN {X 0.121,Y -483.431,Z 539.501,A 0.000,B 0.000,C 90.000,E1 270.172} C_DIS
LIN {X -0.198,Y -481.271,Z 539.498,A 0.000,B 0.000,C 90.000,E1 269.714} C_DIS
LIN {X -0.042,Y -478.397,Z 539.496,A 0.000,B 0.000,C 90.000,E1 269.198} C_DIS
LIN {X 0.091,Y -474.630,Z 539.493,A 0.000,B 0.000,C 90.000,E1 268.682} C_DIS
LIN {X 0.200,Y -469.784,Z 539.490,A 0.000,B 0.000,C 90.000,E1 268.167} C_DIS
LIN {X -0.023,Y -463.882,Z 539.487,A 0.000,B 0.000,C 90.000,E1 267.707} C_DIS
LIN {X -0.220,Y -457.272,Z 539.485,A 0.000,B 0.000,C 90.000,E1 267.306} C_DIS
LIN {X 0.179,Y -450.253,Z 539.483,A 0.000,B 0.000,C 90.000,E1 266.906} C_DIS
LIN {X -0.209,Y -443.168,Z 539.481,A 0.000,B 0.000,C 90.000,E1 266.674} C_DIS
LIN {X -0.214,Y -435.657,Z 539.480,A 0.000,B 0.000,C 90.000,E1 266.445} C_DIS
LIN {X 0.150,Y -427.729,Z 539.479,A 0.000,B 0.000,C 90.000,E1 266.216} C_DIS
LIN {X 0.021,Y -418.880,Z 539.478,A 0.000,B 0.000,C 90.000,E1 266.102} C_DIS
LIN {X -0.066,Y -410.287,Z 539.478,A 0.000,B 0.000,C 90.000,E1 266.045} C_DIS
LIN {X -0.147,Y -405.638,Z 539.478,A 0.000,B 0.000,C 90.000,E1 266.045} C_DIS
LIN {X -0.083,Y -180.921,Z 539.478,A 0.000,B 0.000,C 90.000,E1 266.045} C_DIS
LIN {X -0.026,Y -180.861,Z 539.472,A 0.000,B 0.000,C 90.000,E1 265.008} C_DIS
LIN {X 0.053,Y -178.917,Z 539.443,A 0.000,B 0.000,C 90.000,E1 259.746} C_DIS
LIN {X -0.037,Y -175.963,Z 539.415,A 0.000,B 0.000,C 90.000,E1 254.685} C_DIS
LIN {X 0.079,Y -175.438,Z 539.410,A 0.000,B 0.000,C 90.000,E1 253.795} C_DIS
LIN {X -0.080,Y -172.196,Z 539.386,A 0.000,B 0.000,C 90.000,E1 249.571} C_DIS
LIN {X -0.102,Y -171.669,Z 539.382,A 0.000,B 0.000,C 90.000,E1 248.720} C_DIS
LIN {X 0.041,Y -167.893,Z 539.358,A 0.000,B 0.000,C 90.000,E1 244.357} C_DIS
LIN {X 0.057,Y -166.632,Z 539.348,A 0.000,B 0.000,C 90.000,E1 242.615} C_DIS
LIN {X -0.036,Y -162.618,Z 539.324,A 0.000,B 0.000,C 90.000,E1 238.280} C_DIS
LIN {X 0.023,Y -161.304,Z 539.314,A 0.000,B 0.000,C 90.000,E1 236.501} C_DIS
LIN {X -0.067,Y -157.302,Z 539.289,A 0.000,B 0.000,C 90.000,E1 232.110} C_DIS
LIN {X 0.085,Y -155.278,Z 539.275,A 0.000,B 0.000,C 90.000,E1 229.380} C_DIS
LIN {X 0.014,Y -151.643,Z 539.250,A 0.000,B 0.000,C 90.000,E1 224.919} C_DIS
LIN {X -0.050,Y -150.512,Z 539.240,A 0.000,B 0.000,C 90.000,E1 223.137} C_DIS
LIN {X -0.026,Y -147.236,Z 539.214,A 0.000,B 0.000,C 90.000,E1 218.588} C_DIS
LIN {X 0.059,Y -145.260,Z 539.194,A 0.000,B 0.000,C 90.000,E1 214.898} C_DIS
LIN {X -0.026,Y -142.372,Z 539.163,A 0.000,B 0.000,C 90.000,E1 209.411} C_DIS
LIN {X -0.031,Y -141.757,Z 539.153,A 0.000,B 0.000,C 90.000,E1 207.564} C_DIS
LIN {X 0.021,Y -139.498,Z 539.117,A 0.000,B 0.000,C 90.000,E1 201.046} C_DIS
LIN {X 0.057,Y -139.003,Z 539.101,A 0.000,B 0.000,C 90.000,E1 198.236} C_DIS
LIN {X 0.014,Y -138.339,Z 539.055,A 0.000,B 0.000,C 90.000,E1 189.849} C_DIS
LIN {X 0.036,Y -139.407,Z 539.008,A 0.000,B 0.000,C 90.000,E1 181.432} C_DIS
LIN {X -0.051,Y -141.316,Z 538.972,A 0.000,B 0.000,C 90.000,E1 174.951} C_DIS
LIN {X 0.048,Y -142.676,Z 538.956,A 0.000,B 0.000,C 90.000,E1 172.129} C_DIS
LIN {X 0.028,Y -145.028,Z 538.931,A 0.000,B 0.000,C 90.000,E1 167.521} C_DIS
LIN {X -0.015,Y -147.655,Z 538.910,A 0.000,B 0.000,C 90.000,E1 163.866} C_DIS
LIN {X 0.061,Y -150.292,Z 538.890,A 0.000,B 0.000,C 90.000,E1 160.188} C_DIS
LIN {X -0.067,Y -153.699,Z 538.870,A 0.000,B 0.000,C 90.000,E1 156.613} C_DIS
LIN {X -0.012,Y -157.113,Z 538.850,A 0.000,B 0.000,C 90.000,E1 152.999} C_DIS
LIN {X 0.064,Y -161.255,Z 538.830,A 0.000,B 0.000,C 90.000,E1 149.410} C_DIS
LIN {X -0.008,Y -164.373,Z 538.815,A 0.000,B 0.000,C 90.000,E1 146.786} C_DIS
LIN {X -0.021,Y -169.048,Z 538.796,A 0.000,B 0.000,C 90.000,E1 143.290} C_DIS
LIN {X 0.032,Y -171.610,Z 538.786,A 0.000,B 0.000,C 90.000,E1 141.537} C_DIS
LIN {X 0.080,Y -176.565,Z 538.767,A 0.000,B 0.000,C 90.000,E1 138.081} C_DIS
LIN {X -0.048,Y -180.863,Z 538.753,A 0.000,B 0.000,C 90.000,E1 135.567} C_DIS
LIN {X -0.063,Y -186.276,Z 538.734,A 0.000,B 0.000,C 90.000,E1 132.204} C_DIS
LIN {X -0.003,Y -191.377,Z 538.719,A 0.000,B 0.000,C 90.000,E1 129.402} C_DIS
LIN {X -0.046,Y -192.074,Z 538.717,A 0.000,B 0.000,C 90.000,E1 128.991} C_DIS
LIN {X -0.105,Y -289.022,Z 538.716,A 0.000,B 0.000,C 90.000,E1 128.991} C_DIS
LIN {X 0.154,Y -293.148,Z 538.716,A 0.000,B 0.000,C 90.000,E1 128.830} C_DIS
LIN {X 0.095,Y -295.928,Z 538.715,A 0.000,B 0.000,C 90.000,E1 128.669} C_DIS
LIN {X 0.032,Y -299.651,Z 538.713,A 0.000,B 0.000,C 90.000,E1 128.302} C_DIS
LIN {X 0.017,Y -303.165,Z 538.710,A 0.000,B 0.000,C 90.000,E1 127.729} C_DIS
LIN {X 0.023,Y -304.584,Z 538.708,A 0.000,B 0.000,C 90.000,E1 127.397} C_DIS
LIN {X -0.030,Y -305.701,Z 538.706,A 0.000,B 0.000,C 90.000,E1 127.076} C_DIS
LIN {X 0.128,Y -315.490,Z 538.688,A 0.000,B 0.000,C 90.000,E1 123.785} C_DIS
LIN {X 0.008,Y -325.592,Z 538.672,A 0.000,B 0.000,C 90.000,E1 120.924} C_DIS
LIN {X -0.051,Y -337.030,Z 538.656,A 0.000,B 0.000,C 90.000,E1 118.103} C_DIS
LIN {X -0.095,Y -349.903,Z 538.641,A 0.000,B 0.000,C 90.000,E1 115.335} C_DIS
LIN {X 0.040,Y -362.648,Z 538.627,A 0.000,B 0.000,C 90.000,E1 112.898} C_DIS
LIN {X -0.111,Y -376.711,Z 538.614,A 0.000,B 0.000,C 90.000,E1 110.556} C_DIS
LIN {X -0.053,Y -392.198,Z 538.601,A 0.000,B 0.000,C 90.000,E1 108.236} C_DIS
LIN {X 0.030,Y -409.219,Z 538.589,A 0.000,B 0.000,C 90.000,E1 105.969} C_DIS
LIN {X 0.038,Y -427.900,Z 538.577,A 0.000,B 0.000,C 90.000,E1 103.772} C_DIS
LIN {X -0.179,Y -447.880,Z 538.565,A 0.000,B 0.000,C 90.000,E1 101.715} C_DIS
LIN {X -0.113,Y -468.440,Z 538.554,A 0.000,B 0.000,C 90.000,E1 99.792} C_DIS
LIN {X 0.051,Y -476.278,Z 538.551,A 0.000,B 0.000,C 90.000,E1 99.095} C_DIS
LIN {X 0.151,Y -478.409,Z 538.549,A 0.000,B 0.000,C 90.000,E1 98.859} C_DIS
LIN {X 0.250,Y -480.034,Z 538.548,A 0.000,B 0.000,C 90.000,E1 98.624} C_DIS
LIN {X 0.053,Y -481.424,Z 538.547,A 0.000,B 0.000,C 90.000,E1 98.398} C_DIS
LIN {X -0.075,Y -482.457,Z 538.545,A 0.000,B 0.000,C 90.000,E1 98.163} C_DIS
LIN {X 0.094,Y -483.647,Z 538.543,A 0.000,B 0.000,C 90.000,E1 97.644} C_DIS
LIN {X -0.207,Y -483.827,Z 538.540,A 0.000,B 0.000,C 90.000,E1 97.182} C_DIS
LIN {X -0.022,Y -483.026,Z 538.537,A 0.000,B 0.000,C 90.000,E1 96.663} C_DIS
LIN {X 0.164,Y -481.110,Z 538.534,A 0.000,B 0.000,C 90.000,E1 96.144} C_DIS
LIN {X 0.039,Y -479.616,Z 538.533,A 0.000,B 0.000,C 90.000,E1 95.910} C_DIS
LIN {X 0.100,Y -460.248,Z 538.519,A 0.000,B 0.000,C 90.000,E1 93.383} C_DIS
LIN {X 0.137,Y -449.917,Z 538.510,A 0.000,B 0.000,C 90.000,E1 91.835} C_DIS
LIN {X -0.086,Y -437.598,Z 538.499,A 0.000,B 0.000,C 90.000,E1 89.771} C_DIS
LIN {X 0.003,Y -428.035,Z 538.490,A 0.000,B 0.000,C 90.000,E1 88.165} C_DIS
LIN {X -0.161,Y -413.716,Z 538.476,A 0.000,B 0.000,C 90.000,E1 85.755} C_DIS
LIN {X -0.144,Y -398.051,Z 538.461,A 0.000,B 0.000,C 90.000,E1 82.989} C_DIS
LIN {X 0.149,Y -387.217,Z 538.450,A 0.000,B 0.000,C 90.000,E1 80.971} C_DIS
LIN {X -0.056,Y -376.346,Z 538.439,A 0.000,B 0.000,C 90.000,E1 78.993} C_DIS
LIN {X -0.035,Y -361.306,Z 538.423,A 0.000,B 0.000,C 90.000,E1 76.061} C_DIS
LIN {X -0.143,Y -350.632,Z 538.409,A 0.000,B 0.000,C 90.000,E1 73.685} C_DIS
LIN {X 0.038,Y -340.077,Z 538.394,A 0.000,B 0.000,C 90.000,E1 70.913} C_DIS
LIN {X 0.129,Y -328.577,Z 538.375,A 0.000,B 0.000,C 90.000,E1 67.486} C_DIS
LIN {X 0.108,Y -318.958,Z 538.357,A 0.000,B 0.000,C 90.000,E1 64.332} C_DIS
LIN {X 0.101,Y -311.395,Z 538.343,A 0.000,B 0.000,C 90.000,E1 61.769} C_DIS
LIN {X -0.071,Y -303.912,Z 538.329,A 0.000,B 0.000,C 90.000,E1 59.203} C_DIS
LIN {X 0.064,Y -294.759,Z 538.311,A 0.000,B 0.000,C 90.000,E1 55.881} C_DIS
LIN {X 0.033,Y -287.882,Z 538.296,A 0.000,B 0.000,C 90.000,E1 53.210} C_DIS
LIN {X 0.084,Y -282.689,Z 538.284,A 0.000,B 0.000,C 90.000,E1 51.170} C_DIS
LIN {X -0.021,Y -279.045,Z 538.277,A 0.000,B 0.000,C 90.000,E1 49.828} C_DIS
LIN {X 0.014,Y -275.106,Z 538.269,A 0.000,B 0.000,C 90.000,E1 48.447} C_DIS
LIN {X -0.028,Y -268.666,Z 538.258,A 0.000,B 0.000,C 90.000,E1 46.377} C_DIS
LIN {X 0.102,Y -262.937,Z 538.248,A 0.000,B 0.000,C 90.000,E1 44.595} C_DIS
LIN {X 0.045,Y -253.544,Z 538.232,A 0.000,B 0.000,C 90.000,E1 41.757} C_DIS
LIN {X -0.037,Y -243.507,Z 538.214,A 0.000,B 0.000,C 90.000,E1 38.508} C_DIS
LIN {X 0.113,Y -235.216,Z 538.197,A 0.000,B 0.000,C 90.000,E1 35.518} C_DIS
LIN {X -0.016,Y -227.662,Z 538.181,A 0.000,B 0.000,C 90.000,E1 32.546} C_DIS
LIN {X 0.012,Y -220.976,Z 538.164,A 0.000,B 0.000,C 90.000,E1 29.489} C_DIS
LIN {X -0.043,Y -215.092,Z 538.147,A 0.000,B 0.000,C 90.000,E1 26.411} C_DIS
LIN {X 0.039,Y -210.074,Z 538.129,A 0.000,B 0.000,C 90.000,E1 23.259} C_DIS
LIN {X -0.044,Y -204.845,Z 538.107,A 0.000,B 0.000,C 90.000,E1 19.322} C_DIS
LIN {X 0.027,Y -200.785,Z 538.085,A 0.000,B 0.000,C 90.000,E1 15.300} C_DIS
LIN {X -0.097,Y -197.292,Z 538.058,A 0.000,B 0.000,C 90.000,E1 10.489} C_DIS
LIN {X -0.062,Y -194.847,Z 538.017,A 0.000,B 0.000,C 90.000,E1 3.151} C_DIS
LIN {X 0.070,Y -196.637,Z 537.966,A 0.000,B 0.000,C 90.000,E1 353.799} C_DIS
LIN {X 0.068,Y -199.613,Z 537.939,A 0.000,B 0.000,C 90.000,E1 348.926} C_DIS
LIN {X 0.020,Y -203.877,Z 537.912,A 0.000,B 0.000,C 90.000,E1 344.102} C_DIS
LIN {X -0.012,Y -208.372,Z 537.890,A 0.000,B 0.000,C 90.000,E1 340.115} C_DIS
LIN {X -0.079,Y -213.566,Z 537.868,A 0.000,B 0.000,C 90.000,E1 336.177} C_DIS
LIN {X 0.055,Y -219.360,Z 537.846,A 0.000,B 0.000,C 90.000,E1 332.231} C_DIS
LIN {X -0.098,Y -225.705,Z 537.824,A 0.000,B 0.000,C 90.000,E1 328.408} C_DIS
LIN {X 0.041,Y -232.717,Z 537.803,A 0.000,B 0.000,C 90.000,E1 324.562} C_DIS
LIN {X 0.060,Y -240.151,Z 537.782,A 0.000,B 0.000,C 90.000,E1 320.803} C_DIS
LIN {X -0.120,Y -248.501,Z 537.762,A 0.000,B 0.000,C 90.000,E1 317.148} C_DIS
LIN {X 0.113,Y -257.961,Z 537.742,A 0.000,B 0.000,C 90.000,E1 313.461} C_DIS
LIN {X -0.078,Y -267.666,Z 537.724,A 0.000,B 0.000,C 90.000,E1 310.297} C_DIS
LIN {X 0.002,Y -279.658,Z 537.704,A 0.000,B 0.000,C 90.000,E1 306.790} C_DIS
LIN {X -0.083,Y -290.160,Z 537.689,A 0.000,B 0.000,C 90.000,E1 304.072} C_DIS
LIN {X -0.029,Y -304.544,Z 537.671,A 0.000,B 0.000,C 90.000,E1 300.718} C_DIS
LIN {X -0.026,Y -320.055,Z 537.653,A 0.000,B 0.000,C 90.000,E1 297.462} C_DIS
LIN {X 0.043,Y -330.170,Z 537.642,A 0.000,B 0.000,C 90.000,E1 295.540} C_DIS
LIN {X -0.156,Y -343.284,Z 537.630,A 0.000,B 0.000,C 90.000,E1 293.387} C_DIS
LIN {X 0.024,Y -359.883,Z 537.616,A 0.000,B 0.000,C 90.000,E1 290.918} C_DIS
LIN {X 0.152,Y -382.856,Z 537.600,A 0.000,B 0.000,C 90.000,E1 287.946} C_DIS
LIN {X -0.026,Y -399.770,Z 537.589,A 0.000,B 0.000,C 90.000,E1 285.969} C_DIS
LIN {X 0.035,Y -417.078,Z 537.578,A 0.000,B 0.000,C 90.000,E1 284.008} C_DIS
LIN {X 0.026,Y -429.118,Z 537.570,A 0.000,B 0.000,C 90.000,E1 282.647} C_DIS
LIN {X 0.091,Y -440.579,Z 537.563,A 0.000,B 0.000,C 90.000,E1 281.299} C_DIS
LIN {X -0.217,Y -447.156,Z 537.558,A 0.000,B 0.000,C 90.000,E1 280.546} C_DIS
LIN {X -0.221,Y -455.261,Z 537.553,A 0.000,B 0.000,C 90.000,E1 279.500} C_DIS
LIN {X -0.129,Y -462.708,Z 537.547,A 0.000,B 0.000,C 90.000,E1 278.454} C_DIS
LIN {X 0.211,Y -467.793,Z 537.543,A 0.000,B 0.000,C 90.000,E1 277.644} C_DIS
LIN {X -0.075,Y -473.740,Z 537.537,A 0.000,B 0.000,C 90.000,E1 276.663} C_DIS
LIN {X -0.102,Y -477.631,Z 537.533,A 0.000,B 0.000,C 90.000,E1 275.910} C_DIS
LIN {X -0.151,Y -480.910,Z 537.529,A 0.000,B 0.000,C 90.000,E1 275.163} C_DIS
LIN {X 0.009,Y -482.643,Z 537.526,A 0.000,B 0.000,C 90.000,E1 274.645} C_DIS
LIN {X 0.139,Y -484.091,Z 537.523,A 0.000,B 0.000,C 90.000,E1 274.131} C_DIS
LIN {X -0.169,Y -485.219,Z 537.520,A 0.000,B 0.000,C 90.000,E1 273.669} C_DIS
LIN {X -0.015,Y -486.030,Z 537.518,A 0.000,B 0.000,C 90.000,E1 273.154} C_DIS
LIN {X 0.172,Y -486.523,Z 537.515,A 0.000,B 0.000,C 90.000,E1 272.636} C_DIS
LIN {X -0.144,Y -486.710,Z 537.512,A 0.000,B 0.000,C 90.000,E1 272.178} C_DIS
LIN {X 0.044,Y -486.535,Z 537.509,A 0.000,B 0.000,C 90.000,E1 271.661} C_DIS
LIN {X 0.217,Y -486.004,Z 537.507,A 0.000,B 0.000,C 90.000,E1 271.146} C_DIS
LIN {X -0.095,Y -484.999,Z 537.504,A 0.000,B 0.000,C 90.000,E1 270.688} C_DIS
LIN {X 0.077,Y -483.418,Z 537.501,A 0.000,B 0.000,C 90.000,E1 270.172} C_DIS
LIN {X 0.241,Y -481.263,Z 537.498,A 0.000,B 0.000,C 90.000,E1 269.656} C_DIS
LIN {X 0.077,Y -479.960,Z 537.497,A 0.000,B 0.000,C 90.000,E1 269.427} C_DIS
LIN {X 0.221,Y -476.639,Z 537.494,A 0.000,B 0.000,C 90.000,E1 268.912} C_DIS
LIN {X -0.132,Y -472.327,Z 537.491,A 0.000,B 0.000,C 90.000,E1 268.453} C_DIS
LIN {X 0.074,Y -466.989,Z 537.489,A 0.000,B 0.000,C 90.000,E1 267.936} C_DIS
LIN {X 0.140,Y -460.845,Z 537.486,A 0.000,B 0.000,C 90.000,E1 267.478} C_DIS
LIN {X -0.165,Y -454.132,Z 537.484,A 0.000,B 0.000,C 90.000,E1 267.135} C_DIS
LIN {X 0.075,Y -447.142,Z 537.482,A 0.000,B 0.000,C 90.000,E1 266.788} C_DIS
LIN {X -0.159,Y -439.819,Z 537.481,A 0.000,B 0.000,C 90.000,E1 266.560} C_DIS
LIN {X -0.004,Y -432.319,Z 537.480,A 0.000,B 0.000,C 90.000,E1 266.331} C_DIS
LIN {X 0.088,Y -424.074,Z 537.479,A 0.000,B 0.000,C 90.000,E1 266.159} C_DIS
LIN {X 0.088,Y -414.186,Z 537.478,A 0.000,B 0.000,C 90.000,E1 266.045} C_DIS
LIN {X -0.165,Y -404.938,Z 537.478,A 0.000,B 0.000,C 90.000,E1 266.045} C_DIS
LIN {X -0.092,Y -180.920,Z 537.478,A 0.000,B 0.000,C 90.000,E1 266.045} C_DIS
LIN {X -0.035,Y -180.861,Z 537.472,A 0.000,B 0.000,C 90.000,E1 265.008} C_DIS
LIN {X 0.045,Y -178.916,Z 537.443,A 0.000,B 0.000,C 90.000,E1 259.746} C_DIS
LIN {X -0.045,Y -175.961,Z 537.415,A 0.000,B 0.000,C 90.000,E1 254.685} C_DIS
LIN {X 0.070,Y -175.436,Z 537.410,A 0.000,B 0.000,C 90.000,E1 253.795} C_DIS
LIN {X 0.072,Y -172.194,Z 537.386,A 0.000,B 0.000,C 90.000,E1 249.518} C_DIS
LIN {X 0.049,Y -171.666,Z 537.382,A 0.000,B 0.000,C 90.000,E1 248.666} C_DIS
LIN {X 0.032,Y -167.891,Z 537.358,A 0.000,B 0.000,C 90.000,E1 244.357} C_DIS
LIN {X 0.047,Y -166.629,Z 537.348,A 0.000,B 0.000,C 90.000,E1 242.615} C_DIS
LIN {X 0.041,Y -162.616,Z 537.324,A 0.000,B 0.000,C 90.000,E1 238.250} C_DIS
LIN {X 0.014,Y -161.302,Z 537.314,A 0.000,B 0.000,C 90.000,E1 236.501} C_DIS
LIN {X 0.048,Y -157.300,Z 537.289,A 0.000,B 0.000,C 90.000,E1 232.065} C_DIS
LIN {X 0.078,Y -155.275,Z 537.274,A 0.000,B 0.000,C 90.000,E1 229.380} C_DIS
LIN {X 0.005,Y -151.641,Z 537.250,A 0.000,B 0.000,C 90.000,E1 224.919} C_DIS
LIN {X 0.052,Y -150.510,Z 537.240,A 0.000,B 0.000,C 90.000,E1 223.095} C_DIS
LIN {X -0.034,Y -147.235,Z 537.214,A 0.000,B 0.000,C 90.000,E1 218.588} C_DIS
LIN {X 0.051,Y -145.257,Z 537.194,A 0.000,B 0.000,C 90.000,E1 214.898} C_DIS
LIN {X -0.034,Y -142.370,Z 537.163,A 0.000,B 0.000,C 90.000,E1 209.411} C_DIS
LIN {X 0.088,Y -141.755,Z 537.153,A 0.000,B 0.000,C 90.000,E1 207.513} C_DIS
LIN {X 0.013,Y -139.497,Z 537.117,A 0.000,B 0.000,C 90.000,E1 201.046} C_DIS
LIN {X 0.050,Y -139.003,Z 537.101,A 0.000,B 0.000,C 90.000,E1 198.236} C_DIS
LIN {X 0.006,Y -138.339,Z 537.055,A 0.000,B 0.000,C 90.000,E1 189.849} C_DIS
LIN {X 0.028,Y -139.408,Z 537.008,A 0.000,B 0.000,C 90.000,E1 181.432} C_DIS
LIN {X -0.059,Y -141.318,Z 536.972,A 0.000,B 0.000,C 90.000,E1 174.951} C_DIS
LIN {X 0.040,Y -142.677,Z 536.956,A 0.000,B 0.000,C 90.000,E1 172.129} C_DIS
LIN {X 0.020,Y -145.030,Z 536.931,A 0.000,B 0.000,C 90.000,E1 167.521} C_DIS
LIN {X -0.023,Y -147.657,Z 536.910,A 0.000,B 0.000,C 90.000,E1 163.866} C_DIS
LIN {X 0.054,Y -150.295,Z 536.890,A 0.000,B 0.000,C 90.000,E1 160.188} C_DIS
LIN {X -0.076,Y -153.702,Z 536.870,A 0.000,B 0.000,C 90.000,E1 156.613} C_DIS
LIN {X -0.021,Y -157.116,Z 536.850,A 0.000,B 0.000,C 90.000,E1 152.999} C_DIS
LIN {X 0.055,Y -161.259,Z 536.830,A 0.000,B 0.000,C 90.000,E1 149.410} C_DIS
LIN {X -0.017,Y -164.378,Z 536.815,A 0.000,B 0.000,C 90.000,E1 146.786} C_DIS
LIN {X -0.031,Y -169.052,Z 536.796,A 0.000,B 0.000,C 90.000,E1 143.290} C_DIS
LIN {X 0.023,Y -171.613,Z 536.786,A 0.000,B 0.000,C 90.000,E1 141.537} C_DIS
LIN {X 0.070,Y -176.569,Z 536.767,A 0.000,B 0.000,C 90.000,E1 138.081} C_DIS
LIN {X -0.057,Y -180.868,Z 536.753,A 0.000,B 0.000,C 90.000,E1 135.567} C_DIS
LIN {X 0.065,Y -186.281,Z 536.734,A 0.000,B 0.000,C 90.000,E1 132.162} C_DIS
LIN {X -0.015,Y -191.383,Z 536.719,A 0.000,B 0.000,C 90.000,E1 129.402} C_DIS
LIN {X 0.014,Y -192.105,Z 536.716,A 0.000,B 0.000,C 90.000,E1 128.955} C_DIS
LIN {X -0.014,Y -288.784,Z 536.716,A 0.000,B 0.000,C 90.000,E1 128.955} C_DIS
LIN {X 0.139,Y -292.816,Z 536.716,A 0.000,B 0.000,C 90.000,E1 128.830} C_DIS
LIN {X -0.020,Y -295.994,Z 536.715,A 0.000,B 0.000,C 90.000,E1 128.669} C_DIS
LIN {X -0.032,Y -299.629,Z 536.713,A 0.000,B 0.000,C 90.000,E1 128.302} C_DIS
LIN {X -0.044,Y -303.159,Z 536.710,A 0.000,B 0.000,C 90.000,E1 127.729} C_DIS
LIN {X 0.146,Y -304.588,Z 536.708,A 0.000,B 0.000,C 90.000,E1 127.363} C_DIS
LIN {X -0.092,Y -305.710,Z 536.706,A 0.000,B 0.000,C 90.000,E1 127.076} C_DIS
LIN {X 0.063,Y -315.507,Z 536.688,A 0.000,B 0.000,C 90.000,E1 123.785} C_DIS
LIN {X -0.057,Y -325.613,Z 536.672,A 0.000,B 0.000,C 90.000,E1 120.924} C_DIS
LIN {X -0.117,Y -337.057,Z 536.656,A 0.000,B 0.000,C 90.000,E1 118.103} C_DIS
LIN {X 0.153,Y -349.936,Z 536.641,A 0.000,B 0.000,C 90.000,E1 115.283} C_DIS
LIN {X -0.030,Y -362.685,Z 536.627,A 0.000,B 0.000,C 90.000,E1 112.898} C_DIS
LIN {X -0.184,Y -376.756,Z 536.614,A 0.000,B 0.000,C 90.000,E1 110.556} C_DIS
LIN {X -0.126,Y -392.248,Z 536.601,A 0.000,B 0.000,C 90.000,E1 108.236} C_DIS
LIN {X -0.046,Y -409.276,Z 536.589,A 0.000,B 0.000,C 90.000,E1 105.969} C_DIS
LIN {X -0.039,Y -427.966,Z 536.576,A 0.000,B 0.000,C 90.000,E1 103.772} C_DIS
LIN {X 0.184,Y -447.949,Z 536.565,A 0.000,B 0.000,C 90.000,E1 101.658} C_DIS
LIN {X -0.188,Y -468.513,Z 536.554,A 0.000,B 0.000,C 90.000,E1 99.792} C_DIS
LIN {X -0.022,Y -476.354,Z 536.551,A 0.000,B 0.000,C 90.000,E1 99.095} C_DIS
LIN {X 0.081,Y -478.500,Z 536.549,A 0.000,B 0.000,C 90.000,E1 98.859} C_DIS
LIN {X 0.182,Y -480.135,Z 536.548,A 0.000,B 0.000,C 90.000,E1 98.624} C_DIS
LIN {X -0.015,Y -481.536,Z 536.547,A 0.000,B 0.000,C 90.000,E1 98.398} C_DIS
LIN {X -0.143,Y -482.577,Z 536.545,A 0.000,B 0.000,C 90.000,E1 98.163} C_DIS
LIN {X 0.027,Y -483.780,Z 536.542,A 0.000,B 0.000,C 90.000,E1 97.644} C_DIS
LIN {X 0.206,Y -483.972,Z 536.540,A 0.000,B 0.000,C 90.000,E1 97.125} C_DIS
LIN {X -0.088,Y -483.184,Z 536.537,A 0.000,B 0.000,C 90.000,E1 96.663} C_DIS
LIN {X 0.099,Y -481.284,Z 536.534,A 0.000,B 0.000,C 90.000,E1 96.144} C_DIS
LIN {X -0.025,Y -479.800,Z 536.533,A 0.000,B 0.000,C 90.000,E1 95.910} C_DIS
LIN {X 0.097,Y -469.922,Z 536.526,A 0.000,B 0.000,C 90.000,E1 94.645} C_DIS
LIN {X -0.143,Y -458.594,Z 536.517,A 0.000,B 0.000,C 90.000,E1 93.151} C_DIS
LIN {X 0.083,Y -450.020,Z 536.510,A 0.000,B 0.000,C 90.000,E1 91.835} C_DIS
LIN {X -0.134,Y -437.665,Z 536.499,A 0.000,B 0.000,C 90.000,E1 89.771} C_DIS
LIN {X -0.043,Y -428.089,Z 536.490,A 0.000,B 0.000,C 90.000,E1 88.165} C_DIS
LIN {X 0.208,Y -413.760,Z 536.476,A 0.000,B 0.000,C 90.000,E1 85.698} C_DIS
LIN {X 0.210,Y -398.094,Z 536.461,A 0.000,B 0.000,C 90.000,E1 82.932} C_DIS
LIN {X 0.110,Y -387.240,Z 536.450,A 0.000,B 0.000,C 90.000,E1 80.971} C_DIS
LIN {X -0.094,Y -376.351,Z 536.439,A 0.000,B 0.000,C 90.000,E1 78.993} C_DIS
LIN {X -0.071,Y -361.286,Z 536.422,A 0.000,B 0.000,C 90.000,E1 76.061} C_DIS
LIN {X -0.149,Y -349.376,Z 536.408,A 0.000,B 0.000,C 90.000,E1 73.378} C_DIS
LIN {X 0.008,Y -338.980,Z 536.392,A 0.000,B 0.000,C 90.000,E1 70.604} C_DIS
LIN {X 0.096,Y -328.571,Z 536.375,A 0.000,B 0.000,C 90.000,E1 67.486} C_DIS
LIN {X 0.076,Y -318.964,Z 536.357,A 0.000,B 0.000,C 90.000,E1 64.332} C_DIS
LIN {X 0.091,Y -313.306,Z 536.347,A 0.000,B 0.000,C 90.000,E1 62.410} C_DIS
LIN {X -0.184,Y -305.774,Z 536.332,A 0.000,B 0.000,C 90.000,E1 59.871} C_DIS
LIN {X 0.015,Y -296.491,Z 536.314,A 0.000,B 0.000,C 90.000,E1 56.548} C_DIS
LIN {X 0.003,Y -287.817,Z 536.296,A 0.000,B 0.000,C 90.000,E1 53.210} C_DIS
LIN {X 0.053,Y -282.608,Z 536.284,A 0.000,B 0.000,C 90.000,E1 51.170} C_DIS
LIN {X -0.053,Y -278.959,Z 536.277,A 0.000,B 0.000,C 90.000,E1 49.828} C_DIS
LIN {X -0.020,Y -275.012,Z 536.269,A 0.000,B 0.000,C 90.000,E1 48.447} C_DIS
LIN {X -0.061,Y -268.564,Z 536.258,A 0.000,B 0.000,C 90.000,E1 46.377} C_DIS
LIN {X 0.068,Y -262.816,Z 536.248,A 0.000,B 0.000,C 90.000,E1 44.595} C_DIS
LIN {X 0.008,Y -253.422,Z 536.232,A 0.000,B 0.000,C 90.000,E1 41.757} C_DIS
LIN {X 0.115,Y -243.371,Z 536.214,A 0.000,B 0.000,C 90.000,E1 38.463} C_DIS
LIN {X 0.073,Y -235.094,Z 536.197,A 0.000,B 0.000,C 90.000,E1 35.518} C_DIS
LIN {X -0.057,Y -227.550,Z 536.181,A 0.000,B 0.000,C 90.000,E1 32.546} C_DIS
LIN {X 0.077,Y -220.872,Z 536.164,A 0.000,B 0.000,C 90.000,E1 29.461} C_DIS
LIN {X 0.105,Y -215.009,Z 536.147,A 0.000,B 0.000,C 90.000,E1 26.360} C_DIS
LIN {X -0.007,Y -210.001,Z 536.129,A 0.000,B 0.000,C 90.000,E1 23.259} C_DIS
LIN {X 0.103,Y -204.799,Z 536.107,A 0.000,B 0.000,C 90.000,E1 19.268} C_DIS
LIN {X -0.020,Y -200.764,Z 536.085,A 0.000,B 0.000,C 90.000,E1 15.300} C_DIS
LIN {X 0.049,Y -197.246,Z 536.058,A 0.000,B 0.000,C 90.000,E1 10.433} C_DIS
LIN {X 0.083,Y -194.809,Z 536.017,A 0.000,B 0.000,C 90.000,E1 3.094} C_DIS
LIN {X 0.068,Y -196.573,Z 535.966,A 0.000,B 0.000,C 90.000,E1 353.799} C_DIS
LIN {X 0.063,Y -199.537,Z 535.939,A 0.000,B 0.000,C 90.000,E1 348.926} C_DIS
LIN {X 0.012,Y -203.785,Z 535.912,A 0.000,B 0.000,C 90.000,E1 344.102} C_DIS
LIN {X -0.023,Y -208.299,Z 535.889,A 0.000,B 0.000,C 90.000,E1 340.115} C_DIS
LIN {X -0.092,Y -213.491,Z 535.867,A 0.000,B 0.000,C 90.000,E1 336.177} C_DIS
LIN {X 0.038,Y -219.285,Z 535.846,A 0.000,B 0.000,C 90.000,E1 332.231} C_DIS
LIN {X -0.117,Y -225.635,Z 535.824,A 0.000,B 0.000,C 90.000,E1 328.408} C_DIS
LIN {X 0.019,Y -232.636,Z 535.803,A 0.000,B 0.000,C 90.000,E1 324.562} C_DIS
LIN {X 0.034,Y -240.093,Z 535.782,A 0.000,B 0.000,C 90.000,E1 320.803} C_DIS
LIN {X 0.033,Y -248.457,Z 535.762,A 0.000,B 0.000,C 90.000,E1 317.106} C_DIS
LIN {X 0.083,Y -257.948,Z 535.742,A 0.000,B 0.000,C 90.000,E1 313.461} C_DIS
LIN {X 0.094,Y -267.658,Z 535.724,A 0.000,B 0.000,C 90.000,E1 310.253} C_DIS
LIN {X -0.033,Y -279.651,Z 535.704,A 0.000,B 0.000,C 90.000,E1 306.790} C_DIS
LIN {X 0.020,Y -291.553,Z 535.687,A 0.000,B 0.000,C 90.000,E1 303.706} C_DIS
LIN {X -0.044,Y -306.029,Z 535.669,A 0.000,B 0.000,C 90.000,E1 300.384} C_DIS
LIN {X 0.003,Y -321.653,Z 535.651,A 0.000,B 0.000,C 90.000,E1 297.129} C_DIS
LIN {X 0.099,Y -331.938,Z 535.640,A 0.000,B 0.000,C 90.000,E1 295.207} C_DIS
LIN {X 0.115,Y -343.277,Z 535.630,A 0.000,B 0.000,C 90.000,E1 293.334} C_DIS
LIN {X -0.022,Y -359.874,Z 535.616,A 0.000,B 0.000,C 90.000,E1 290.918} C_DIS
LIN {X 0.103,Y -382.875,Z 535.600,A 0.000,B 0.000,C 90.000,E1 287.946} C_DIS
LIN {X -0.076,Y -399.791,Z 535.589,A 0.000,B 0.000,C 90.000,E1 285.969} C_DIS
LIN {X -0.018,Y -417.116,Z 535.578,A 0.000,B 0.000,C 90.000,E1 284.008} C_DIS
LIN {X -0.026,Y -429.200,Z 535.570,A 0.000,B 0.000,C 90.000,E1 282.647} C_DIS
LIN {X 0.038,Y -440.675,Z 535.563,A 0.000,B 0.000,C 90.000,E1 281.299} C_DIS
LIN {X 0.169,Y -447.285,Z 535.558,A 0.000,B 0.000,C 90.000,E1 280.489} C_DIS
LIN {X 0.176,Y -455.413,Z 535.553,A 0.000,B 0.000,C 90.000,E1 279.443} C_DIS
LIN {X -0.180,Y -462.871,Z 535.547,A 0.000,B 0.000,C 90.000,E1 278.454} C_DIS
LIN {X 0.161,Y -467.945,Z 535.543,A 0.000,B 0.000,C 90.000,E1 277.644} C_DIS
LIN {X 0.088,Y -472.501,Z 535.538,A 0.000,B 0.000,C 90.000,E1 276.891} C_DIS
LIN {X -0.151,Y -477.757,Z 535.533,A 0.000,B 0.000,C 90.000,E1 275.910} C_DIS
LIN {X -0.198,Y -481.012,Z 535.529,A 0.000,B 0.000,C 90.000,E1 275.163} C_DIS
LIN {X -0.038,Y -482.745,Z 535.526,A 0.000,B 0.000,C 90.000,E1 274.645} C_DIS
LIN {X 0.092,Y -484.196,Z 535.523,A 0.000,B 0.000,C 90.000,E1 274.131} C_DIS
LIN {X -0.215,Y -485.294,Z 535.520,A 0.000,B 0.000,C 90.000,E1 273.669} C_DIS
LIN {X -0.061,Y -486.090,Z 535.517,A 0.000,B 0.000,C 90.000,E1 273.154} C_DIS
LIN {X 0.128,Y -486.607,Z 535.515,A 0.000,B 0.000,C 90.000,E1 272.636} C_DIS
LIN {X -0.189,Y -486.769,Z 535.512,A 0.000,B 0.000,C 90.000,E1 272.178} C_DIS
LIN {X -0.001,Y -486.605,Z 535.509,A 0.000,B 0.000,C 90.000,E1 271.661} C_DIS
LIN {X 0.173,Y -486.002,Z 535.506,A 0.000,B 0.000,C 90.000,E1 271.146} C_DIS
LIN {X -0.138,Y -484.992,Z 535.504,A 0.000,B 0.000,C 90.000,E1 270.688} C_DIS
LIN {X 0.033,Y -483.420,Z 535.501,A 0.000,B 0.000,C 90.000,E1 270.172} C_DIS
LIN {X 0.197,Y -481.271,Z 535.498,A 0.000,B 0.000,C 90.000,E1 269.656} C_DIS
LIN {X -0.128,Y -478.396,Z 535.495,A 0.000,B 0.000,C 90.000,E1 269.198} C_DIS
LIN {X 0.005,Y -474.574,Z 535.493,A 0.000,B 0.000,C 90.000,E1 268.682} C_DIS
LIN {X 0.130,Y -469.691,Z 535.490,A 0.000,B 0.000,C 90.000,E1 268.165} C_DIS
LIN {X 0.016,Y -466.893,Z 535.489,A 0.000,B 0.000,C 90.000,E1 267.936} C_DIS
LIN {X -0.097,Y -463.755,Z 535.487,A 0.000,B 0.000,C 90.000,E1 267.707} C_DIS
LIN {X 0.058,Y -460.651,Z 535.486,A 0.000,B 0.000,C 90.000,E1 267.478} C_DIS
LIN {X 0.205,Y -453.963,Z 535.484,A 0.000,B 0.000,C 90.000,E1 267.078} C_DIS
LIN {X 0.019,Y -446.929,Z 535.482,A 0.000,B 0.000,C 90.000,E1 266.788} C_DIS
LIN {X -0.193,Y -439.791,Z 535.481,A 0.000,B 0.000,C 90.000,E1 266.560} C_DIS
LIN {X -0.013,Y -432.288,Z 535.480,A 0.000,B 0.000,C 90.000,E1 266.331} C_DIS
LIN {X 0.083,Y -424.305,Z 535.479,A 0.000,B 0.000,C 90.000,E1 266.159} C_DIS
LIN {X 0.079,Y -414.553,Z 535.478,A 0.000,B 0.000,C 90.000,E1 266.045} C_DIS
LIN {X -0.187,Y -403.686,Z 535.478,A 0.000,B 0.000,C 90.000,E1 266.045} C_DIS
LIN {X 0.077,Y -180.921,Z 535.478,A 0.000,B 0.000,C 90.000,E1 265.988} C_DIS
LIN {X -0.047,Y -180.860,Z 535.472,A 0.000,B 0.000,C 90.000,E1 265.008} C_DIS
LIN {X 0.032,Y -178.915,Z 535.443,A 0.000,B 0.000,C 90.000,E1 259.746} C_DIS
LIN {X -0.057,Y -175.959,Z 535.415,A 0.000,B 0.000,C 90.000,E1 254.685} C_DIS
LIN {X 0.059,Y -175.433,Z 535.410,A 0.000,B 0.000,C 90.000,E1 253.795} C_DIS
LIN {X 0.061,Y -172.192,Z 535.386,A 0.000,B 0.000,C 90.000,E1 249.518} C_DIS
LIN {X 0.037,Y -171.664,Z 535.382,A 0.000,B 0.000,C 90.000,E1 248.666} C_DIS
LIN {X 0.021,Y -167.889,Z 535.358,A 0.000,B 0.000,C 90.000,E1 244.357} C_DIS
LIN {X 0.037,Y -166.626,Z 535.348,A 0.000,B 0.000,C 90.000,E1 242.615} C_DIS
LIN {X 0.030,Y -162.612,Z 535.324,A 0.000,B 0.000,C 90.000,E1 238.250} C_DIS
LIN {X 0.004,Y -161.298,Z 535.314,A 0.000,B 0.000,C 90.000,E1 236.501} C_DIS
LIN {X 0.038,Y -157.296,Z 535.289,A 0.000,B 0.000,C 90.000,E1 232.065} C_DIS
LIN {X 0.066,Y -155.271,Z 535.274,A 0.000,B 0.000,C 90.000,E1 229.380} C_DIS
LIN {X -0.005,Y -151.639,Z 535.250,A 0.000,B 0.000,C 90.000,E1 224.919} C_DIS
LIN {X 0.042,Y -150.508,Z 535.240,A 0.000,B 0.000,C 90.000,E1 223.095} C_DIS
LIN {X 0.071,Y -147.232,Z 535.214,A 0.000,B 0.000,C 90.000,E1 218.543} C_DIS
LIN {X 0.040,Y -145.255,Z 535.194,A 0.000,B 0.000,C 90.000,E1 214.898} C_DIS
LIN {X -0.044,Y -142.369,Z 535.163,A 0.000,B 0.000,C 90.000,E1 209.411} C_DIS
LIN {X 0.077,Y -141.754,Z 535.153,A 0.000,B 0.000,C 90.000,E1 207.513} C_DIS
LIN {X 0.002,Y -139.496,Z 535.117,A 0.000,B 0.000,C 90.000,E1 201.046} C_DIS
LIN {X 0.040,Y -139.001,Z 535.101,A 0.000,B 0.000,C 90.000,E1 198.236} C_DIS
LIN {X -0.004,Y -138.338,Z 535.055,A 0.000,B 0.000,C 90.000,E1 189.849} C_DIS
LIN {X 0.018,Y -139.409,Z 535.008,A 0.000,B 0.000,C 90.000,E1 181.432} C_DIS
LIN {X -0.069,Y -141.319,Z 534.972,A 0.000,B 0.000,C 90.000,E1 174.951} C_DIS
LIN {X 0.030,Y -142.678,Z 534.956,A 0.000,B 0.000,C 90.000,E1 172.129} C_DIS
LIN {X 0.009,Y -145.033,Z 534.931,A 0.000,B 0.000,C 90.000,E1 167.521} C_DIS
LIN {X -0.034,Y -147.659,Z 534.910,A 0.000,B 0.000,C 90.000,E1 163.866} C_DIS
LIN {X 0.042,Y -150.298,Z 534.890,A 0.000,B 0.000,C 90.000,E1 160.188} C_DIS
LIN {X -0.087,Y -153.707,Z 534.870,A 0.000,B 0.000,C 90.000,E1 156.613} C_DIS
LIN {X -0.032,Y -157.120,Z 534.850,A 0.000,B 0.000,C 90.000,E1 152.999} C_DIS
LIN {X 0.044,Y -161.264,Z 534.830,A 0.000,B 0.000,C 90.000,E1 149.410} C_DIS
LIN {X -0.029,Y -164.382,Z 534.815,A 0.000,B 0.000,C 90.000,E1 146.786} C_DIS
LIN {X -0.041,Y -169.058,Z 534.796,A 0.000,B 0.000,C 90.000,E1 143.290} C_DIS
LIN {X 0.011,Y -171.619,Z 534.786,A 0.000,B 0.000,C 90.000,E1 141.537} C_DIS
LIN {X 0.059,Y -176.575,Z 534.767,A 0.000,B 0.000,C 90.000,E1 138.081} C_DIS
LIN {X -0.068,Y -180.873,Z 534.753,A 0.000,B 0.000,C 90.000,E1 135.567} C_DIS
LIN {X 0.053,Y -186.287,Z 534.734,A 0.000,B 0.000,C 90.000,E1 132.162} C_DIS
LIN {X -0.028,Y -191.390,Z 534.719,A 0.000,B 0.000,C 90.000,E1 129.402} C_DIS
LIN {X 0.076,Y -192.148,Z 534.716,A 0.000,B 0.000,C 90.000,E1 128.910} C_DIS
LIN {X 0.080,Y -289.505,Z 534.716,A 0.000,B 0.000,C 90.000,E1 128.910} C_DIS
LIN {X 0.121,Y -292.433,Z 534.716,A 0.000,B 0.000,C 90.000,E1 128.830} C_DIS
LIN {X -0.063,Y -295.869,Z 534.715,A 0.000,B 0.000,C 90.000,E1 128.669} C_DIS
LIN {X 0.015,Y -299.429,Z 534.713,A 0.000,B 0.000,C 90.000,E1 128.302} C_DIS
LIN {X 0.071,Y -302.989,Z 534.710,A 0.000,B 0.000,C 90.000,E1 127.729} C_DIS
LIN {X -0.167,Y -304.462,Z 534.708,A 0.000,B 0.000,C 90.000,E1 127.443} C_DIS
LIN {X 0.022,Y -305.621,Z 534.706,A 0.000,B 0.000,C 90.000,E1 127.076} C_DIS
LIN {X -0.023,Y -316.477,Z 534.686,A 0.000,B 0.000,C 90.000,E1 123.499} C_DIS
LIN {X 0.153,Y -326.719,Z 534.670,A 0.000,B 0.000,C 90.000,E1 120.590} C_DIS
LIN {X 0.134,Y -338.304,Z 534.654,A 0.000,B 0.000,C 90.000,E1 117.769} C_DIS
LIN {X -0.028,Y -351.342,Z 534.639,A 0.000,B 0.000,C 90.000,E1 115.027} C_DIS
LIN {X -0.185,Y -364.242,Z 534.626,A 0.000,B 0.000,C 90.000,E1 112.642} C_DIS
LIN {X 0.044,Y -378.473,Z 534.613,A 0.000,B 0.000,C 90.000,E1 110.248} C_DIS
LIN {X 0.028,Y -394.140,Z 534.600,A 0.000,B 0.000,C 90.000,E1 107.946} C_DIS
LIN {X -0.113,Y -411.356,Z 534.587,A 0.000,B 0.000,C 90.000,E1 105.717} C_DIS
LIN {X -0.173,Y -430.249,Z 534.575,A 0.000,B 0.000,C 90.000,E1 103.536} C_DIS
LIN {X 0.197,Y -450.319,Z 534.564,A 0.000,B 0.000,C 90.000,E1 101.422} C_DIS
LIN {X -0.020,Y -470.943,Z 534.553,A 0.000,B 0.000,C 90.000,E1 99.557} C_DIS
LIN {X 0.091,Y -476.177,Z 534.551,A 0.000,B 0.000,C 90.000,E1 99.095} C_DIS
LIN {X 0.198,Y -478.400,Z 534.549,A 0.000,B 0.000,C 90.000,E1 98.859} C_DIS
LIN {X -0.170,Y -480.087,Z 534.548,A 0.000,B 0.000,C 90.000,E1 98.681} C_DIS
LIN {X 0.107,Y -481.536,Z 534.547,A 0.000,B 0.000,C 90.000,E1 98.398} C_DIS
LIN {X -0.021,Y -482.616,Z 534.545,A 0.000,B 0.000,C 90.000,E1 98.163} C_DIS
LIN {X 0.150,Y -483.882,Z 534.543,A 0.000,B 0.000,C 90.000,E1 97.644} C_DIS
LIN {X -0.151,Y -484.130,Z 534.540,A 0.000,B 0.000,C 90.000,E1 97.182} C_DIS
LIN {X 0.035,Y -483.400,Z 534.537,A 0.000,B 0.000,C 90.000,E1 96.663} C_DIS
LIN {X 0.223,Y -481.572,Z 534.534,A 0.000,B 0.000,C 90.000,E1 96.144} C_DIS
LIN {X 0.099,Y -480.136,Z 534.533,A 0.000,B 0.000,C 90.000,E1 95.910} C_DIS
LIN {X -0.099,Y -472.293,Z 534.527,A 0.000,B 0.000,C 90.000,E1 94.935} C_DIS
LIN {X 0.172,Y -460.723,Z 534.519,A 0.000,B 0.000,C 90.000,E1 93.383} C_DIS
LIN {X 0.215,Y -450.279,Z 534.510,A 0.000,B 0.000,C 90.000,E1 91.835} C_DIS
LIN {X -0.175,Y -439.448,Z 534.500,A 0.000,B 0.000,C 90.000,E1 90.057} C_DIS
LIN {X -0.064,Y -429.893,Z 534.491,A 0.000,B 0.000,C 90.000,E1 88.453} C_DIS
LIN {X 0.123,Y -417.112,Z 534.479,A 0.000,B 0.000,C 90.000,E1 86.274} C_DIS
LIN {X -0.025,Y -406.020,Z 534.469,A 0.000,B 0.000,C 90.000,E1 84.375} C_DIS
LIN {X 0.069,Y -393.630,Z 534.456,A 0.000,B 0.000,C 90.000,E1 82.129} C_DIS
LIN {X -0.001,Y -382.762,Z 534.445,A 0.000,B 0.000,C 90.000,E1 80.151} C_DIS
LIN {X 0.148,Y -368.799,Z 534.431,A 0.000,B 0.000,C 90.000,E1 77.521} C_DIS
LIN {X 0.116,Y -360.005,Z 534.421,A 0.000,B 0.000,C 90.000,E1 75.755} C_DIS
LIN {X -0.086,Y -348.255,Z 534.406,A 0.000,B 0.000,C 90.000,E1 73.087} C_DIS
LIN {X 0.140,Y -339.083,Z 534.392,A 0.000,B 0.000,C 90.000,E1 70.604} C_DIS
LIN {X -0.077,Y -328.655,Z 534.375,A 0.000,B 0.000,C 90.000,E1 67.539} C_DIS
LIN {X 0.066,Y -319.051,Z 534.358,A 0.000,B 0.000,C 90.000,E1 64.357} C_DIS
LIN {X -0.076,Y -311.480,Z 534.343,A 0.000,B 0.000,C 90.000,E1 61.820} C_DIS
LIN {X 0.025,Y -303.939,Z 534.329,A 0.000,B 0.000,C 90.000,E1 59.203} C_DIS
LIN {X -0.086,Y -294.730,Z 534.311,A 0.000,B 0.000,C 90.000,E1 55.928} C_DIS
LIN {X 0.125,Y -287.817,Z 534.296,A 0.000,B 0.000,C 90.000,E1 53.210} C_DIS
LIN {X 0.173,Y -282.605,Z 534.284,A 0.000,B 0.000,C 90.000,E1 51.170} C_DIS
LIN {X 0.066,Y -278.945,Z 534.277,A 0.000,B 0.000,C 90.000,E1 49.828} C_DIS
LIN {X -0.084,Y -275.000,Z 534.269,A 0.000,B 0.000,C 90.000,E1 48.485} C_DIS
LIN {X 0.082,Y -270.741,Z 534.262,A 0.000,B 0.000,C 90.000,E1 47.067} C_DIS
LIN {X 0.066,Y -265.145,Z 534.252,A 0.000,B 0.000,C 90.000,E1 45.324} C_DIS
LIN {X -0.011,Y -258.096,Z 534.240,A 0.000,B 0.000,C 90.000,E1 43.218} C_DIS
LIN {X -0.142,Y -246.612,Z 534.220,A 0.000,B 0.000,C 90.000,E1 39.644} C_DIS
LIN {X 0.025,Y -237.065,Z 534.202,A 0.000,B 0.000,C 90.000,E1 36.297} C_DIS
LIN {X 0.071,Y -229.343,Z 534.185,A 0.000,B 0.000,C 90.000,E1 33.293} C_DIS
LIN {X 0.057,Y -222.441,Z 534.168,A 0.000,B 0.000,C 90.000,E1 30.256} C_DIS
LIN {X 0.033,Y -216.369,Z 534.151,A 0.000,B 0.000,C 90.000,E1 27.180} C_DIS
LIN {X -0.046,Y -211.160,Z 534.134,A 0.000,B 0.000,C 90.000,E1 24.079} C_DIS
LIN {X -0.015,Y -205.736,Z 534.112,A 0.000,B 0.000,C 90.000,E1 20.120} C_DIS
LIN {X -0.046,Y -201.490,Z 534.090,A 0.000,B 0.000,C 90.000,E1 16.134} C_DIS
LIN {X -0.060,Y -197.710,Z 534.063,A 0.000,B 0.000,C 90.000,E1 11.299} C_DIS
LIN {X 0.051,Y -195.020,Z 534.027,A 0.000,B 0.000,C 90.000,E1 4.759} C_DIS
LIN {X 0.065,Y -196.508,Z 533.966,A 0.000,B 0.000,C 90.000,E1 353.799} C_DIS
LIN {X 0.056,Y -200.083,Z 533.934,A 0.000,B 0.000,C 90.000,E1 348.117} C_DIS
LIN {X -0.080,Y -204.528,Z 533.907,A 0.000,B 0.000,C 90.000,E1 343.323} C_DIS
LIN {X -0.095,Y -209.187,Z 533.885,A 0.000,B 0.000,C 90.000,E1 339.337} C_DIS
LIN {X 0.020,Y -214.524,Z 533.863,A 0.000,B 0.000,C 90.000,E1 335.357} C_DIS
LIN {X 0.093,Y -220.444,Z 533.841,A 0.000,B 0.000,C 90.000,E1 331.435} C_DIS
LIN {X 0.097,Y -226.886,Z 533.820,A 0.000,B 0.000,C 90.000,E1 327.582} C_DIS
LIN {X 0.091,Y -234.012,Z 533.799,A 0.000,B 0.000,C 90.000,E1 323.783} C_DIS
LIN {X -0.039,Y -241.652,Z 533.778,A 0.000,B 0.000,C 90.000,E1 320.070} C_DIS
LIN {X -0.012,Y -250.213,Z 533.758,A 0.000,B 0.000,C 90.000,E1 316.377} C_DIS
LIN {X -0.075,Y -260.005,Z 533.738,A 0.000,B 0.000,C 90.000,E1 312.771} C_DIS
LIN {X 0.066,Y -271.121,Z 533.718,A 0.000,B 0.000,C 90.000,E1 309.197} C_DIS
LIN {X 0.097,Y -283.468,Z 533.699,A 0.000,B 0.000,C 90.000,E1 305.724} C_DIS
LIN {X 0.100,Y -297.228,Z 533.680,A 0.000,B 0.000,C 90.000,E1 302.339} C_DIS
LIN {X -0.095,Y -312.114,Z 533.661,A 0.000,B 0.000,C 90.000,E1 299.077} C_DIS
LIN {X 0.061,Y -326.635,Z 533.645,A 0.000,B 0.000,C 90.000,E1 296.155} C_DIS
LIN {X 0.109,Y -337.472,Z 533.635,A 0.000,B 0.000,C 90.000,E1 294.259} C_DIS
LIN {X -0.210,Y -351.393,Z 533.623,A 0.000,B 0.000,C 90.000,E1 292.153} C_DIS
LIN {X 0.112,Y -366.544,Z 533.611,A 0.000,B 0.000,C 90.000,E1 289.993} C_DIS
LIN {X 0.182,Y -385.281,Z 533.598,A 0.000,B 0.000,C 90.000,E1 287.638} C_DIS
LIN {X 0.128,Y -402.167,Z 533.587,A 0.000,B 0.000,C 90.000,E1 285.662} C_DIS
LIN {X 0.015,Y -417.034,Z 533.578,A 0.000,B 0.000,C 90.000,E1 284.008} C_DIS
LIN {X 0.007,Y -429.168,Z 533.570,A 0.000,B 0.000,C 90.000,E1 282.647} C_DIS
LIN {X 0.070,Y -440.702,Z 533.563,A 0.000,B 0.000,C 90.000,E1 281.299} C_DIS
LIN {X -0.237,Y -447.319,Z 533.558,A 0.000,B 0.000,C 90.000,E1 280.546} C_DIS
LIN {X -0.239,Y -455.474,Z 533.553,A 0.000,B 0.000,C 90.000,E1 279.500} C_DIS
LIN {X 0.101,Y -461.165,Z 533.548,A 0.000,B 0.000,C 90.000,E1 278.681} C_DIS
LIN {X -0.095,Y -466.419,Z 533.544,A 0.000,B 0.000,C 90.000,E1 277.936} C_DIS
LIN {X -0.186,Y -471.113,Z 533.540,A 0.000,B 0.000,C 90.000,E1 277.182} C_DIS
LIN {X 0.035,Y -476.611,Z 533.534,A 0.000,B 0.000,C 90.000,E1 276.144} C_DIS
LIN {X 0.030,Y -480.054,Z 533.530,A 0.000,B 0.000,C 90.000,E1 275.391} C_DIS
LIN {X -0.157,Y -481.093,Z 533.529,A 0.000,B 0.000,C 90.000,E1 275.163} C_DIS
LIN {X 0.004,Y -482.828,Z 533.526,A 0.000,B 0.000,C 90.000,E1 274.645} C_DIS
LIN {X 0.134,Y -484.267,Z 533.523,A 0.000,B 0.000,C 90.000,E1 274.131} C_DIS
LIN {X -0.172,Y -485.375,Z 533.520,A 0.000,B 0.000,C 90.000,E1 273.669} C_DIS
LIN {X -0.017,Y -486.189,Z 533.518,A 0.000,B 0.000,C 90.000,E1 273.154} C_DIS
LIN {X 0.171,Y -486.709,Z 533.515,A 0.000,B 0.000,C 90.000,E1 272.636} C_DIS
LIN {X -0.145,Y -486.866,Z 533.512,A 0.000,B 0.000,C 90.000,E1 272.178} C_DIS
LIN {X 0.044,Y -486.680,Z 533.509,A 0.000,B 0.000,C 90.000,E1 271.661} C_DIS
LIN {X 0.218,Y -486.097,Z 533.507,A 0.000,B 0.000,C 90.000,E1 271.146} C_DIS
LIN {X -0.092,Y -485.075,Z 533.504,A 0.000,B 0.000,C 90.000,E1 270.688} C_DIS
LIN {X 0.078,Y -483.514,Z 533.501,A 0.000,B 0.000,C 90.000,E1 270.172} C_DIS
LIN {X -0.238,Y -481.344,Z 533.498,A 0.000,B 0.000,C 90.000,E1 269.714} C_DIS
LIN {X -0.081,Y -478.455,Z 533.495,A 0.000,B 0.000,C 90.000,E1 269.198} C_DIS
LIN {X 0.052,Y -474.632,Z 533.493,A 0.000,B 0.000,C 90.000,E1 268.682} C_DIS
LIN {X -0.129,Y -472.336,Z 533.491,A 0.000,B 0.000,C 90.000,E1 268.453} C_DIS
LIN {X 0.069,Y -466.964,Z 533.489,A 0.000,B 0.000,C 90.000,E1 267.936} C_DIS
LIN {X -0.039,Y -463.845,Z 533.487,A 0.000,B 0.000,C 90.000,E1 267.707} C_DIS
LIN {X -0.196,Y -457.292,Z 533.485,A 0.000,B 0.000,C 90.000,E1 267.306} C_DIS
LIN {X -0.230,Y -450.364,Z 533.483,A 0.000,B 0.000,C 90.000,E1 266.963} C_DIS
LIN {X -0.182,Y -443.214,Z 533.481,A 0.000,B 0.000,C 90.000,E1 266.674} C_DIS
LIN {X -0.207,Y -435.846,Z 533.480,A 0.000,B 0.000,C 90.000,E1 266.445} C_DIS
LIN {X 0.143,Y -428.087,Z 533.479,A 0.000,B 0.000,C 90.000,E1 266.216} C_DIS
LIN {X -0.017,Y -419.573,Z 533.478,A 0.000,B 0.000,C 90.000,E1 266.102} C_DIS
LIN {X -0.114,Y -410.406,Z 533.478,A 0.000,B 0.000,C 90.000,E1 266.045} C_DIS
LIN {X -0.203,Y -405.558,Z 533.478,A 0.000,B 0.000,C 90.000,E1 266.045} C_DIS
LIN {X 0.070,Y -180.921,Z 533.478,A 0.000,B 0.000,C 90.000,E1 265.988} C_DIS
LIN {X -0.055,Y -180.860,Z 533.472,A 0.000,B 0.000,C 90.000,E1 265.008} C_DIS
LIN {X 0.025,Y -178.914,Z 533.443,A 0.000,B 0.000,C 90.000,E1 259.746} C_DIS
LIN {X -0.066,Y -175.958,Z 533.415,A 0.000,B 0.000,C 90.000,E1 254.685} C_DIS
LIN {X 0.051,Y -175.431,Z 533.410,A 0.000,B 0.000,C 90.000,E1 253.795} C_DIS
LIN {X 0.053,Y -172.189,Z 533.386,A 0.000,B 0.000,C 90.000,E1 249.518} C_DIS
LIN {X 0.030,Y -171.662,Z 533.382,A 0.000,B 0.000,C 90.000,E1 248.666} C_DIS
LIN {X 0.014,Y -167.887,Z 533.358,A 0.000,B 0.000,C 90.000,E1 244.357} C_DIS
LIN {X 0.029,Y -166.624,Z 533.348,A 0.000,B 0.000,C 90.000,E1 242.615} C_DIS
LIN {X 0.021,Y -162.610,Z 533.324,A 0.000,B 0.000,C 90.000,E1 238.250} C_DIS
LIN {X -0.004,Y -161.296,Z 533.314,A 0.000,B 0.000,C 90.000,E1 236.501} C_DIS
LIN {X 0.030,Y -157.294,Z 533.289,A 0.000,B 0.000,C 90.000,E1 232.065} C_DIS
LIN {X 0.053,Y -156.011,Z 533.279,A 0.000,B 0.000,C 90.000,E1 230.275} C_DIS
LIN {X 0.013,Y -152.270,Z 533.255,A 0.000,B 0.000,C 90.000,E1 225.810} C_DIS
LIN {X 0.035,Y -150.506,Z 533.240,A 0.000,B 0.000,C 90.000,E1 223.095} C_DIS
LIN {X 0.065,Y -147.230,Z 533.214,A 0.000,B 0.000,C 90.000,E1 218.543} C_DIS
LIN {X 0.033,Y -145.254,Z 533.194,A 0.000,B 0.000,C 90.000,E1 214.898} C_DIS
LIN {X -0.051,Y -142.368,Z 533.163,A 0.000,B 0.000,C 90.000,E1 209.411} C_DIS
LIN {X 0.070,Y -141.753,Z 533.153,A 0.000,B 0.000,C 90.000,E1 207.513} C_DIS
LIN {X -0.004,Y -139.496,Z 533.117,A 0.000,B 0.000,C 90.000,E1 201.046} C_DIS
LIN {X 0.033,Y -139.000,Z 533.101,A 0.000,B 0.000,C 90.000,E1 198.236} C_DIS
LIN {X -0.011,Y -138.338,Z 533.055,A 0.000,B 0.000,C 90.000,E1 189.849} C_DIS
LIN {X 0.011,Y -139.410,Z 533.008,A 0.000,B 0.000,C 90.000,E1 181.432} C_DIS
LIN {X 0.065,Y -141.320,Z 532.972,A 0.000,B 0.000,C 90.000,E1 174.894} C_DIS
LIN {X 0.023,Y -142.679,Z 532.956,A 0.000,B 0.000,C 90.000,E1 172.129} C_DIS
LIN {X 0.003,Y -145.035,Z 532.931,A 0.000,B 0.000,C 90.000,E1 167.521} C_DIS
LIN {X -0.040,Y -147.661,Z 532.910,A 0.000,B 0.000,C 90.000,E1 163.866} C_DIS
LIN {X 0.036,Y -150.300,Z 532.890,A 0.000,B 0.000,C 90.000,E1 160.188} C_DIS
LIN {X -0.094,Y -153.709,Z 532.870,A 0.000,B 0.000,C 90.000,E1 156.613} C_DIS
LIN {X -0.039,Y -157.123,Z 532.850,A 0.000,B 0.000,C 90.000,E1 152.999} C_DIS
LIN {X 0.037,Y -161.267,Z 532.830,A 0.000,B 0.000,C 90.000,E1 149.410} C_DIS
LIN {X -0.036,Y -164.386,Z 532.815,A 0.000,B 0.000,C 90.000,E1 146.786} C_DIS
LIN {X -0.050,Y -169.062,Z 532.796,A 0.000,B 0.000,C 90.000,E1 143.290} C_DIS
LIN {X 0.003,Y -171.622,Z 532.786,A 0.000,B 0.000,C 90.000,E1 141.537} C_DIS
LIN {X 0.050,Y -176.580,Z 532.767,A 0.000,B 0.000,C 90.000,E1 138.081} C_DIS
LIN {X -0.076,Y -180.878,Z 532.753,A 0.000,B 0.000,C 90.000,E1 135.567} C_DIS
LIN {X 0.044,Y -186.292,Z 532.734,A 0.000,B 0.000,C 90.000,E1 132.162} C_DIS
LIN {X -0.039,Y -191.396,Z 532.719,A 0.000,B 0.000,C 90.000,E1 129.402} C_DIS
LIN {X 0.041,Y -192.166,Z 532.716,A 0.000,B 0.000,C 90.000,E1 128.910} C_DIS
LIN {X 0.026,Y -288.866,Z 532.716,A 0.000,B 0.000,C 90.000,E1 128.910} C_DIS
LIN {X 0.107,Y -292.114,Z 532.716,A 0.000,B 0.000,C 90.000,E1 128.830} C_DIS
LIN {X 0.059,Y -295.364,Z 532.715,A 0.000,B 0.000,C 90.000,E1 128.669} C_DIS
LIN {X -0.143,Y -298.906,Z 532.713,A 0.000,B 0.000,C 90.000,E1 128.382} C_DIS
LIN {X 0.082,Y -302.504,Z 532.710,A 0.000,B 0.000,C 90.000,E1 127.810} C_DIS
LIN {X -0.156,Y -304.087,Z 532.708,A 0.000,B 0.000,C 90.000,E1 127.523} C_DIS
LIN {X 0.030,Y -305.332,Z 532.706,A 0.000,B 0.000,C 90.000,E1 127.156} C_DIS
LIN {X -0.020,Y -316.191,Z 532.687,A 0.000,B 0.000,C 90.000,E1 123.579} C_DIS
LIN {X 0.152,Y -326.398,Z 532.671,A 0.000,B 0.000,C 90.000,E1 120.669} C_DIS
LIN {X 0.131,Y -337.945,Z 532.655,A 0.000,B 0.000,C 90.000,E1 117.847} C_DIS
LIN {X 0.116,Y -350.941,Z 532.639,A 0.000,B 0.000,C 90.000,E1 115.079} C_DIS
LIN {X -0.053,Y -363.800,Z 532.626,A 0.000,B 0.000,C 90.000,E1 112.695} C_DIS
LIN {X 0.164,Y -377.989,Z 532.613,A 0.000,B 0.000,C 90.000,E1 110.301} C_DIS
LIN {X 0.134,Y -393.609,Z 532.600,A 0.000,B 0.000,C 90.000,E1 108.000} C_DIS
LIN {X -0.130,Y -410.776,Z 532.588,A 0.000,B 0.000,C 90.000,E1 105.788} C_DIS
LIN {X -0.094,Y -429.615,Z 532.575,A 0.000,B 0.000,C 90.000,E1 103.592} C_DIS
LIN {X -0.209,Y -449.667,Z 532.564,A 0.000,B 0.000,C 90.000,E1 101.535} C_DIS
LIN {X -0.028,Y -470.276,Z 532.553,A 0.000,B 0.000,C 90.000,E1 99.613} C_DIS
LIN {X 0.198,Y -477.900,Z 532.550,A 0.000,B 0.000,C 90.000,E1 98.916} C_DIS
LIN {X -0.222,Y -479.721,Z 532.548,A 0.000,B 0.000,C 90.000,E1 98.746} C_DIS
LIN {X 0.126,Y -481.300,Z 532.547,A 0.000,B 0.000,C 90.000,E1 98.454} C_DIS
LIN {X -0.003,Y -482.482,Z 532.546,A 0.000,B 0.000,C 90.000,E1 98.219} C_DIS
LIN {X 0.166,Y -483.916,Z 532.543,A 0.000,B 0.000,C 90.000,E1 97.701} C_DIS
LIN {X -0.137,Y -484.313,Z 532.540,A 0.000,B 0.000,C 90.000,E1 97.239} C_DIS
LIN {X 0.049,Y -483.733,Z 532.537,A 0.000,B 0.000,C 90.000,E1 96.720} C_DIS
LIN {X -0.242,Y -482.085,Z 532.535,A 0.000,B 0.000,C 90.000,E1 96.258} C_DIS
LIN {X 0.115,Y -480.768,Z 532.533,A 0.000,B 0.000,C 90.000,E1 95.967} C_DIS
LIN {X -0.235,Y -477.037,Z 532.530,A 0.000,B 0.000,C 90.000,E1 95.511} C_DIS
LIN {X 0.203,Y -461.383,Z 532.519,A 0.000,B 0.000,C 90.000,E1 93.440} C_DIS
LIN {X -0.195,Y -450.840,Z 532.511,A 0.000,B 0.000,C 90.000,E1 91.949} C_DIS
LIN {X 0.051,Y -438.379,Z 532.499,A 0.000,B 0.000,C 90.000,E1 89.828} C_DIS
LIN {X -0.134,Y -427.176,Z 532.489,A 0.000,B 0.000,C 90.000,E1 87.993} C_DIS
LIN {X 0.001,Y -414.417,Z 532.477,A 0.000,B 0.000,C 90.000,E1 85.812} C_DIS
LIN {X -0.054,Y -400.259,Z 532.463,A 0.000,B 0.000,C 90.000,E1 83.337} C_DIS
LIN {X -0.100,Y -390.975,Z 532.454,A 0.000,B 0.000,C 90.000,E1 81.659} C_DIS
LIN {X 0.096,Y -380.083,Z 532.443,A 0.000,B 0.000,C 90.000,E1 79.634} C_DIS
LIN {X -0.130,Y -364.693,Z 532.426,A 0.000,B 0.000,C 90.000,E1 76.756} C_DIS
LIN {X 0.155,Y -354.989,Z 532.415,A 0.000,B 0.000,C 90.000,E1 74.629} C_DIS
LIN {X -0.015,Y -346.177,Z 532.403,A 0.000,B 0.000,C 90.000,E1 72.543} C_DIS
LIN {X 0.162,Y -337.232,Z 532.389,A 0.000,B 0.000,C 90.000,E1 70.061} C_DIS
LIN {X 0.015,Y -326.936,Z 532.372,A 0.000,B 0.000,C 90.000,E1 66.975} C_DIS
LIN {X -0.064,Y -319.293,Z 532.358,A 0.000,B 0.000,C 90.000,E1 64.460} C_DIS
LIN {X -0.041,Y -313.628,Z 532.347,A 0.000,B 0.000,C 90.000,E1 62.538} C_DIS
LIN {X -0.038,Y -306.048,Z 532.333,A 0.000,B 0.000,C 90.000,E1 59.950} C_DIS
LIN {X -0.036,Y -298.534,Z 532.318,A 0.000,B 0.000,C 90.000,E1 57.327} C_DIS
LIN {X 0.010,Y -289.706,Z 532.300,A 0.000,B 0.000,C 90.000,E1 53.989} C_DIS
LIN {X -0.078,Y -284.520,Z 532.289,A 0.000,B 0.000,C 90.000,E1 51.984} C_DIS
LIN {X 0.087,Y -279.094,Z 532.277,A 0.000,B 0.000,C 90.000,E1 49.908} C_DIS
LIN {X -0.062,Y -275.178,Z 532.270,A 0.000,B 0.000,C 90.000,E1 48.566} C_DIS
LIN {X 0.106,Y -270.914,Z 532.262,A 0.000,B 0.000,C 90.000,E1 47.148} C_DIS
LIN {X 0.091,Y -265.340,Z 532.252,A 0.000,B 0.000,C 90.000,E1 45.405} C_DIS
LIN {X 0.061,Y -257.122,Z 532.239,A 0.000,B 0.000,C 90.000,E1 42.933} C_DIS
LIN {X -0.097,Y -245.683,Z 532.219,A 0.000,B 0.000,C 90.000,E1 39.358} C_DIS
LIN {X 0.065,Y -237.200,Z 532.202,A 0.000,B 0.000,C 90.000,E1 36.377} C_DIS
LIN {X -0.075,Y -229.487,Z 532.186,A 0.000,B 0.000,C 90.000,E1 33.420} C_DIS
LIN {X 0.109,Y -222.568,Z 532.169,A 0.000,B 0.000,C 90.000,E1 30.335} C_DIS
LIN {X 0.090,Y -216.479,Z 532.152,A 0.000,B 0.000,C 90.000,E1 27.257} C_DIS
LIN {X 0.018,Y -211.250,Z 532.134,A 0.000,B 0.000,C 90.000,E1 24.155} C_DIS
LIN {X 0.115,Y -206.796,Z 532.117,A 0.000,B 0.000,C 90.000,E1 20.972} C_DIS
LIN {X -0.077,Y -202.320,Z 532.095,A 0.000,B 0.000,C 90.000,E1 17.040} C_DIS
LIN {X -0.004,Y -198.266,Z 532.068,A 0.000,B 0.000,C 90.000,E1 12.187} C_DIS
LIN {X 0.048,Y -195.443,Z 532.036,A 0.000,B 0.000,C 90.000,E1 6.486} C_DIS
LIN {X 0.063,Y -196.438,Z 531.966,A 0.000,B 0.000,C 90.000,E1 353.799} C_DIS
LIN {X 0.050,Y -199.996,Z 531.934,A 0.000,B 0.000,C 90.000,E1 348.117} C_DIS
LIN {X -0.089,Y -204.437,Z 531.907,A 0.000,B 0.000,C 90.000,E1 343.323} C_DIS
LIN {X -0.034,Y -209.090,Z 531.885,A 0.000,B 0.000,C 90.000,E1 339.316} C_DIS
LIN {X 0.004,Y -214.449,Z 531.863,A 0.000,B 0.000,C 90.000,E1 335.357} C_DIS
LIN {X 0.074,Y -220.348,Z 531.841,A 0.000,B 0.000,C 90.000,E1 331.435} C_DIS
LIN {X 0.075,Y -226.803,Z 531.820,A 0.000,B 0.000,C 90.000,E1 327.582} C_DIS
LIN {X 0.065,Y -233.931,Z 531.799,A 0.000,B 0.000,C 90.000,E1 323.783} C_DIS
LIN {X -0.067,Y -241.590,Z 531.778,A 0.000,B 0.000,C 90.000,E1 320.070} C_DIS
LIN {X -0.044,Y -250.184,Z 531.758,A 0.000,B 0.000,C 90.000,E1 316.377} C_DIS
LIN {X -0.109,Y -260.005,Z 531.737,A 0.000,B 0.000,C 90.000,E1 312.771} C_DIS
LIN {X 0.030,Y -271.114,Z 531.718,A 0.000,B 0.000,C 90.000,E1 309.197} C_DIS
LIN {X 0.059,Y -283.472,Z 531.699,A 0.000,B 0.000,C 90.000,E1 305.724} C_DIS
LIN {X 0.061,Y -297.224,Z 531.680,A 0.000,B 0.000,C 90.000,E1 302.339} C_DIS
LIN {X -0.137,Y -312.097,Z 531.661,A 0.000,B 0.000,C 90.000,E1 299.077} C_DIS
LIN {X 0.017,Y -326.616,Z 531.645,A 0.000,B 0.000,C 90.000,E1 296.155} C_DIS
LIN {X -0.055,Y -335.576,Z 531.637,A 0.000,B 0.000,C 90.000,E1 294.591} C_DIS
LIN {X 0.050,Y -349.331,Z 531.625,A 0.000,B 0.000,C 90.000,E1 292.408} C_DIS
LIN {X -0.008,Y -364.292,Z 531.613,A 0.000,B 0.000,C 90.000,E1 290.301} C_DIS
LIN {X 0.128,Y -385.306,Z 531.598,A 0.000,B 0.000,C 90.000,E1 287.638} C_DIS
LIN {X 0.082,Y -402.182,Z 531.587,A 0.000,B 0.000,C 90.000,E1 285.662} C_DIS
LIN {X -0.033,Y -417.059,Z 531.578,A 0.000,B 0.000,C 90.000,E1 284.008} C_DIS
LIN {X -0.043,Y -429.223,Z 531.570,A 0.000,B 0.000,C 90.000,E1 282.647} C_DIS
LIN {X 0.021,Y -440.815,Z 531.563,A 0.000,B 0.000,C 90.000,E1 281.299} C_DIS
LIN {X 0.154,Y -447.449,Z 531.558,A 0.000,B 0.000,C 90.000,E1 280.489} C_DIS
LIN {X 0.162,Y -455.632,Z 531.553,A 0.000,B 0.000,C 90.000,E1 279.443} C_DIS
LIN {X 0.053,Y -461.311,Z 531.548,A 0.000,B 0.000,C 90.000,E1 278.681} C_DIS
LIN {X -0.143,Y -466.573,Z 531.544,A 0.000,B 0.000,C 90.000,E1 277.936} C_DIS
LIN {X -0.232,Y -471.254,Z 531.540,A 0.000,B 0.000,C 90.000,E1 277.182} C_DIS
LIN {X 0.192,Y -475.473,Z 531.536,A 0.000,B 0.000,C 90.000,E1 276.372} C_DIS
LIN {X 0.126,Y -479.140,Z 531.531,A 0.000,B 0.000,C 90.000,E1 275.625} C_DIS
LIN {X -0.202,Y -481.214,Z 531.529,A 0.000,B 0.000,C 90.000,E1 275.163} C_DIS
LIN {X -0.040,Y -482.954,Z 531.526,A 0.000,B 0.000,C 90.000,E1 274.645} C_DIS
LIN {X 0.091,Y -484.376,Z 531.523,A 0.000,B 0.000,C 90.000,E1 274.131} C_DIS
LIN {X -0.215,Y -485.495,Z 531.520,A 0.000,B 0.000,C 90.000,E1 273.669} C_DIS
LIN {X -0.059,Y -486.314,Z 531.517,A 0.000,B 0.000,C 90.000,E1 273.154} C_DIS
LIN {X 0.130,Y -486.807,Z 531.515,A 0.000,B 0.000,C 90.000,E1 272.636} C_DIS
LIN {X -0.186,Y -486.956,Z 531.512,A 0.000,B 0.000,C 90.000,E1 272.178} C_DIS
LIN {X 0.005,Y -486.768,Z 531.509,A 0.000,B 0.000,C 90.000,E1 271.661} C_DIS
LIN {X 0.179,Y -486.158,Z 531.506,A 0.000,B 0.000,C 90.000,E1 271.146} C_DIS
LIN {X -0.131,Y -485.143,Z 531.504,A 0.000,B 0.000,C 90.000,E1 270.688} C_DIS
LIN {X 0.040,Y -483.582,Z 531.501,A 0.000,B 0.000,C 90.000,E1 270.172} C_DIS
LIN {X 0.205,Y -481.392,Z 531.498,A 0.000,B 0.000,C 90.000,E1 269.656} C_DIS
LIN {X -0.124,Y -478.460,Z 531.495,A 0.000,B 0.000,C 90.000,E1 269.198} C_DIS
LIN {X 0.181,Y -476.700,Z 531.494,A 0.000,B 0.000,C 90.000,E1 268.912} C_DIS
LIN {X -0.171,Y -472.301,Z 531.491,A 0.000,B 0.000,C 90.000,E1 268.453} C_DIS
LIN {X 0.136,Y -469.756,Z 531.490,A 0.000,B 0.000,C 90.000,E1 268.165} C_DIS
LIN {X 0.006,Y -466.908,Z 531.489,A 0.000,B 0.000,C 90.000,E1 267.936} C_DIS
LIN {X 0.056,Y -460.666,Z 531.486,A 0.000,B 0.000,C 90.000,E1 267.478} C_DIS
LIN {X 0.213,Y -453.983,Z 531.484,A 0.000,B 0.000,C 90.000,E1 267.078} C_DIS
LIN {X 0.018,Y -446.920,Z 531.482,A 0.000,B 0.000,C 90.000,E1 266.788} C_DIS
LIN {X -0.189,Y -439.859,Z 531.481,A 0.000,B 0.000,C 90.000,E1 266.560} C_DIS
LIN {X -0.033,Y -432.394,Z 531.480,A 0.000,B 0.000,C 90.000,E1 266.331} C_DIS
LIN {X 0.033,Y -424.316,Z 531.479,A 0.000,B 0.000,C 90.000,E1 266.159} C_DIS
LIN {X 0.028,Y -414.551,Z 531.478,A 0.000,B 0.000,C 90.000,E1 266.045} C_DIS
LIN {X 0.163,Y -405.511,Z 531.478,A 0.000,B 0.000,C 90.000,E1 265.988} C_DIS
LIN {X 0.053,Y -180.921,Z 531.478,A 0.000,B 0.000,C 90.000,E1 265.988} C_DIS
LIN {X -0.071,Y -180.858,Z 531.472,A 0.000,B 0.000,C 90.000,E1 265.008} C_DIS
LIN {X 0.008,Y -178.912,Z 531.443,A 0.000,B 0.000,C 90.000,E1 259.746} C_DIS
LIN {X 0.088,Y -175.957,Z 531.415,A 0.000,B 0.000,C 90.000,E1 254.629} C_DIS
LIN {X 0.035,Y -175.426,Z 531.410,A 0.000,B 0.000,C 90.000,E1 253.795} C_DIS
LIN {X 0.037,Y -172.186,Z 531.386,A 0.000,B 0.000,C 90.000,E1 249.518} C_DIS
LIN {X 0.014,Y -171.658,Z 531.382,A 0.000,B 0.000,C 90.000,E1 248.666} C_DIS
LIN {X -0.003,Y -167.882,Z 531.358,A 0.000,B 0.000,C 90.000,E1 244.357} C_DIS
LIN {X 0.013,Y -166.619,Z 531.348,A 0.000,B 0.000,C 90.000,E1 242.615} C_DIS
LIN {X 0.007,Y -162.606,Z 531.324,A 0.000,B 0.000,C 90.000,E1 238.250} C_DIS
LIN {X -0.020,Y -161.292,Z 531.314,A 0.000,B 0.000,C 90.000,E1 236.501} C_DIS
LIN {X 0.016,Y -157.290,Z 531.289,A 0.000,B 0.000,C 90.000,E1 232.065} C_DIS
LIN {X 0.038,Y -156.007,Z 531.279,A 0.000,B 0.000,C 90.000,E1 230.275} C_DIS
LIN {X -0.002,Y -152.265,Z 531.255,A 0.000,B 0.000,C 90.000,E1 225.810} C_DIS
LIN {X 0.020,Y -150.503,Z 531.239,A 0.000,B 0.000,C 90.000,E1 223.095} C_DIS
LIN {X 0.049,Y -147.227,Z 531.214,A 0.000,B 0.000,C 90.000,E1 218.543} C_DIS
LIN {X 0.019,Y -145.250,Z 531.194,A 0.000,B 0.000,C 90.000,E1 214.898} C_DIS
LIN {X -0.065,Y -142.366,Z 531.163,A 0.000,B 0.000,C 90.000,E1 209.411} C_DIS
LIN {X 0.056,Y -141.751,Z 531.153,A 0.000,B 0.000,C 90.000,E1 207.513} C_DIS
LIN {X -0.019,Y -139.494,Z 531.117,A 0.000,B 0.000,C 90.000,E1 201.046} C_DIS
LIN {X 0.019,Y -138.999,Z 531.101,A 0.000,B 0.000,C 90.000,E1 198.236} C_DIS
LIN {X -0.024,Y -138.337,Z 531.055,A 0.000,B 0.000,C 90.000,E1 189.849} C_DIS
LIN {X -0.003,Y -139.411,Z 531.008,A 0.000,B 0.000,C 90.000,E1 181.432} C_DIS
LIN {X 0.051,Y -141.323,Z 530.972,A 0.000,B 0.000,C 90.000,E1 174.894} C_DIS
LIN {X 0.008,Y -142.681,Z 530.956,A 0.000,B 0.000,C 90.000,E1 172.129} C_DIS
LIN {X -0.012,Y -145.038,Z 530.931,A 0.000,B 0.000,C 90.000,E1 167.521} C_DIS
LIN {X -0.055,Y -147.664,Z 530.910,A 0.000,B 0.000,C 90.000,E1 163.866} C_DIS
LIN {X 0.020,Y -150.305,Z 530.890,A 0.000,B 0.000,C 90.000,E1 160.188} C_DIS
LIN {X 0.032,Y -153.715,Z 530.870,A 0.000,B 0.000,C 90.000,E1 156.561} C_DIS
LIN {X -0.054,Y -157.129,Z 530.850,A 0.000,B 0.000,C 90.000,E1 152.999} C_DIS
LIN {X 0.021,Y -161.274,Z 530.830,A 0.000,B 0.000,C 90.000,E1 149.410} C_DIS
LIN {X 0.039,Y -164.392,Z 530.815,A 0.000,B 0.000,C 90.000,E1 146.755} C_DIS
LIN {X 0.036,Y -169.069,Z 530.796,A 0.000,B 0.000,C 90.000,E1 143.256} C_DIS
LIN {X -0.013,Y -171.629,Z 530.786,A 0.000,B 0.000,C 90.000,E1 141.537} C_DIS
LIN {X 0.034,Y -176.588,Z 530.767,A 0.000,B 0.000,C 90.000,E1 138.081} C_DIS
LIN {X -0.093,Y -180.887,Z 530.753,A 0.000,B 0.000,C 90.000,E1 135.567} C_DIS
LIN {X 0.028,Y -186.301,Z 530.734,A 0.000,B 0.000,C 90.000,E1 132.162} C_DIS
LIN {X -0.058,Y -191.404,Z 530.719,A 0.000,B 0.000,C 90.000,E1 129.402} C_DIS
LIN {X -0.027,Y -192.199,Z 530.716,A 0.000,B 0.000,C 90.000,E1 128.910} C_DIS
LIN {X -0.076,Y -289.661,Z 530.716,A 0.000,B 0.000,C 90.000,E1 128.910} C_DIS
LIN {X 0.082,Y -291.878,Z 530.716,A 0.000,B 0.000,C 90.000,E1 128.830} C_DIS
LIN {X -0.045,Y -294.942,Z 530.715,A 0.000,B 0.000,C 90.000,E1 128.705} C_DIS
LIN {X 0.052,Y -298.470,Z 530.713,A 0.000,B 0.000,C 90.000,E1 128.382} C_DIS
LIN {X -0.002,Y -302.090,Z 530.711,A 0.000,B 0.000,C 90.000,E1 127.890} C_DIS
LIN {X -0.058,Y -303.768,Z 530.709,A 0.000,B 0.000,C 90.000,E1 127.569} C_DIS
LIN {X -0.057,Y -305.085,Z 530.707,A 0.000,B 0.000,C 90.000,E1 127.237} C_DIS
LIN {X 0.061,Y -315.966,Z 530.687,A 0.000,B 0.000,C 90.000,E1 123.627} C_DIS
LIN {X 0.054,Y -326.144,Z 530.671,A 0.000,B 0.000,C 90.000,E1 120.747} C_DIS
LIN {X 0.185,Y -337.661,Z 530.655,A 0.000,B 0.000,C 90.000,E1 117.897} C_DIS
